  PROC DrawPart23()
    MoveL Offs(pOrigin,99.71,-142.38,-0.00),v40,z0,tcp\WObj:=Plywood;
    MoveL Offs(pOrigin,98.01,-141.25,-0.00),v40,z0,tcp\WObj:=Plywood;
    MoveL Offs(pOrigin,101.27,-145.36,-0.00),v40,fine,tcp\WObj:=Plywood;
    MoveL Offs(pOrigin,101.27,-145.36,-6.00),v60,z5,tcp\WObj:=Plywood;
    MoveL Offs(pOrigin,101.48,-143.34,-6.00),vTravel,z5,tcp\WObj:=Plywood;
    MoveL Offs(pOrigin,101.48,-143.34,-0.00),v60,z0,tcp\WObj:=Plywood;
    MoveL Offs(pOrigin,101.02,-141.85,-0.00),v40,z0,tcp\WObj:=Plywood;
    MoveL Offs(pOrigin,99.39,-139.44,-0.00),v40,z0,tcp\WObj:=Plywood;
    MoveL Offs(pOrigin,99.36,-140.36,-0.00),v40,z0,tcp\WObj:=Plywood;
    MoveL Offs(pOrigin,101.48,-143.34,-0.00),v40,fine,tcp\WObj:=Plywood;
    MoveL Offs(pOrigin,101.48,-143.34,-6.00),v60,z5,tcp\WObj:=Plywood;
    MoveL Offs(pOrigin,99.15,-144.93,-6.00),vTravel,z5,tcp\WObj:=Plywood;
    MoveL Offs(pOrigin,99.15,-144.93,-0.00),v60,z0,tcp\WObj:=Plywood;
    MoveL Offs(pOrigin,97.91,-143.34,-0.00),v40,z0,tcp\WObj:=Plywood;
    MoveL Offs(pOrigin,97.06,-142.95,-0.00),v40,z0,tcp\WObj:=Plywood;
    MoveL Offs(pOrigin,99.15,-144.93,-0.00),v40,fine,tcp\WObj:=Plywood;
    MoveL Offs(pOrigin,99.15,-144.93,-6.00),v60,z5,tcp\WObj:=Plywood;
    MoveL Offs(pOrigin,98.33,-142.70,-6.00),vTravel,z5,tcp\WObj:=Plywood;
    MoveL Offs(pOrigin,98.33,-142.70,-0.00),v60,z0,tcp\WObj:=Plywood;
    MoveL Offs(pOrigin,98.12,-142.17,-0.00),v40,z0,tcp\WObj:=Plywood;
    MoveL Offs(pOrigin,98.33,-142.70,-0.00),v40,fine,tcp\WObj:=Plywood;
    MoveL Offs(pOrigin,98.33,-142.70,-6.00),v60,z5,tcp\WObj:=Plywood;
    MoveL Offs(pOrigin,97.73,-140.68,-6.00),vTravel,z5,tcp\WObj:=Plywood;
    MoveL Offs(pOrigin,97.73,-140.68,-0.00),v60,z0,tcp\WObj:=Plywood;
    MoveL Offs(pOrigin,98.37,-140.79,-0.00),v40,z0,tcp\WObj:=Plywood;
    MoveL Offs(pOrigin,97.73,-140.68,-0.00),v40,fine,tcp\WObj:=Plywood;
    MoveL Offs(pOrigin,97.73,-140.68,-6.00),v60,z5,tcp\WObj:=Plywood;
    MoveL Offs(pOrigin,98.97,-140.33,-6.00),vTravel,z5,tcp\WObj:=Plywood;
    MoveL Offs(pOrigin,98.97,-140.33,-0.00),v60,z0,tcp\WObj:=Plywood;
    MoveL Offs(pOrigin,98.65,-139.87,-0.00),v40,z0,tcp\WObj:=Plywood;
    MoveL Offs(pOrigin,98.97,-140.33,-0.00),v40,fine,tcp\WObj:=Plywood;
    MoveL Offs(pOrigin,98.97,-140.33,-6.00),v60,z5,tcp\WObj:=Plywood;
    MoveL Offs(pOrigin,99.89,-138.98,-6.00),vTravel,z5,tcp\WObj:=Plywood;
    MoveL Offs(pOrigin,99.89,-138.98,-0.00),v60,z0,tcp\WObj:=Plywood;
    MoveL Offs(pOrigin,100.53,-139.62,-0.00),v40,z0,tcp\WObj:=Plywood;
    MoveL Offs(pOrigin,99.43,-137.71,-0.00),v40,z0,tcp\WObj:=Plywood;
    MoveL Offs(pOrigin,99.89,-138.98,-0.00),v40,z0,tcp\WObj:=Plywood;
    MoveL Offs(pOrigin,100.35,-137.95,-0.00),v40,z0,tcp\WObj:=Plywood;
    MoveL Offs(pOrigin,100.14,-137.35,-0.00),v40,z0,tcp\WObj:=Plywood;
    MoveL Offs(pOrigin,100.35,-137.95,-0.00),v40,fine,tcp\WObj:=Plywood;
    MoveL Offs(pOrigin,100.35,-137.95,-6.00),v60,z5,tcp\WObj:=Plywood;
    MoveL Offs(pOrigin,101.41,-137.18,-6.00),vTravel,z5,tcp\WObj:=Plywood;
    MoveL Offs(pOrigin,101.41,-137.18,-0.00),v60,z0,tcp\WObj:=Plywood;
    MoveL Offs(pOrigin,101.84,-137.95,-0.00),v40,z0,tcp\WObj:=Plywood;
    MoveL Offs(pOrigin,101.41,-136.18,-0.00),v40,z0,tcp\WObj:=Plywood;
    MoveL Offs(pOrigin,101.41,-137.18,-0.00),v40,z0,tcp\WObj:=Plywood;
    MoveL Offs(pOrigin,100.88,-136.57,-0.00),v40,z0,tcp\WObj:=Plywood;
    MoveL Offs(pOrigin,100.92,-136.22,-0.00),v40,z0,tcp\WObj:=Plywood;
    MoveL Offs(pOrigin,100.56,-136.04,-0.00),v40,z0,tcp\WObj:=Plywood;
    MoveL Offs(pOrigin,100.88,-136.57,-0.00),v40,z0,tcp\WObj:=Plywood;
    MoveL Offs(pOrigin,100.99,-136.01,-0.00),v40,z0,tcp\WObj:=Plywood;
    MoveL Offs(pOrigin,100.78,-135.58,-0.00),v40,z0,tcp\WObj:=Plywood;
    MoveL Offs(pOrigin,100.99,-136.01,-0.00),v40,z0,tcp\WObj:=Plywood;
    MoveL Offs(pOrigin,100.56,-135.05,-0.00),v40,z0,tcp\WObj:=Plywood;
    MoveL Offs(pOrigin,100.99,-135.26,-0.00),v40,z0,tcp\WObj:=Plywood;
    MoveL Offs(pOrigin,100.56,-135.05,-0.00),v40,fine,tcp\WObj:=Plywood;
    MoveL Offs(pOrigin,100.56,-135.05,-6.00),v60,z5,tcp\WObj:=Plywood;
    MoveL Offs(pOrigin,102.05,-133.99,-6.00),vTravel,z5,tcp\WObj:=Plywood;
    MoveL Offs(pOrigin,102.05,-133.99,-0.00),v60,z0,tcp\WObj:=Plywood;
    MoveL Offs(pOrigin,103.32,-134.34,-0.00),v40,z0,tcp\WObj:=Plywood;
    MoveL Offs(pOrigin,103.93,-134.94,-0.00),v40,z0,tcp\WObj:=Plywood;
    MoveL Offs(pOrigin,103.54,-132.54,-0.00),v40,z0,tcp\WObj:=Plywood;
    MoveL Offs(pOrigin,102.90,-133.17,-0.00),v40,z0,tcp\WObj:=Plywood;
    MoveL Offs(pOrigin,101.84,-133.03,-0.00),v40,z0,tcp\WObj:=Plywood;
    MoveL Offs(pOrigin,101.73,-133.56,-0.00),v40,z0,tcp\WObj:=Plywood;
    MoveL Offs(pOrigin,102.05,-133.99,-0.00),v40,fine,tcp\WObj:=Plywood;
    MoveL Offs(pOrigin,102.05,-133.99,-6.00),v60,z5,tcp\WObj:=Plywood;
    MoveL Offs(pOrigin,103.86,-134.20,-6.00),vTravel,z5,tcp\WObj:=Plywood;
    MoveL Offs(pOrigin,103.86,-134.20,-0.00),v60,z0,tcp\WObj:=Plywood;
    MoveL Offs(pOrigin,104.60,-135.37,-0.00),v40,z0,tcp\WObj:=Plywood;
    MoveL Offs(pOrigin,109.38,-136.86,-0.00),v40,z0,tcp\WObj:=Plywood;
    MoveL Offs(pOrigin,112.14,-137.18,-0.00),v40,z0,tcp\WObj:=Plywood;
    MoveL Offs(pOrigin,116.07,-137.07,-0.00),v40,z0,tcp\WObj:=Plywood;
    MoveL Offs(pOrigin,117.35,-136.68,-0.00),v40,z0,tcp\WObj:=Plywood;
    MoveL Offs(pOrigin,118.41,-135.62,-0.00),v40,z0,tcp\WObj:=Plywood;
    MoveL Offs(pOrigin,120.86,-136.32,-0.00),v40,z0,tcp\WObj:=Plywood;
    MoveL Offs(pOrigin,122.66,-136.25,-0.00),v40,z0,tcp\WObj:=Plywood;
    MoveL Offs(pOrigin,123.51,-137.71,-0.00),v40,z0,tcp\WObj:=Plywood;
    MoveL Offs(pOrigin,126.06,-138.88,-0.00),v40,z0,tcp\WObj:=Plywood;
    MoveL Offs(pOrigin,132.01,-139.94,-0.00),v40,z0,tcp\WObj:=Plywood;
    MoveL Offs(pOrigin,136.48,-139.44,-0.00),v40,z0,tcp\WObj:=Plywood;
    MoveL Offs(pOrigin,137.22,-138.98,-0.00),v40,z0,tcp\WObj:=Plywood;
    MoveL Offs(pOrigin,137.86,-137.60,-0.00),v40,z0,tcp\WObj:=Plywood;
    MoveL Offs(pOrigin,138.07,-133.77,-0.00),v40,z0,tcp\WObj:=Plywood;
    MoveL Offs(pOrigin,137.32,-131.65,-0.00),v40,z0,tcp\WObj:=Plywood;
    MoveL Offs(pOrigin,134.88,-130.48,-0.00),v40,z0,tcp\WObj:=Plywood;
    MoveL Offs(pOrigin,131.91,-129.84,-0.00),v40,z0,tcp\WObj:=Plywood;
    MoveL Offs(pOrigin,127.55,-129.63,-0.00),v40,z0,tcp\WObj:=Plywood;
    MoveL Offs(pOrigin,126.06,-130.02,-0.00),v40,z0,tcp\WObj:=Plywood;
    MoveL Offs(pOrigin,124.89,-131.01,-0.00),v40,z0,tcp\WObj:=Plywood;
    MoveL Offs(pOrigin,123.90,-132.50,-0.00),v40,z0,tcp\WObj:=Plywood;
    MoveL Offs(pOrigin,122.77,-135.48,-0.00),v40,z0,tcp\WObj:=Plywood;
    MoveL Offs(pOrigin,121.71,-135.79,-0.00),v40,z0,tcp\WObj:=Plywood;
    MoveL Offs(pOrigin,119.79,-135.58,-0.00),v40,z0,tcp\WObj:=Plywood;
    MoveL Offs(pOrigin,118.55,-134.94,-0.00),v40,z0,tcp\WObj:=Plywood;
    MoveL Offs(pOrigin,118.20,-131.44,-0.00),v40,z0,tcp\WObj:=Plywood;
    MoveL Offs(pOrigin,117.49,-129.63,-0.00),v40,z0,tcp\WObj:=Plywood;
    MoveL Offs(pOrigin,116.71,-128.78,-0.00),v40,z0,tcp\WObj:=Plywood;
    MoveL Offs(pOrigin,112.89,-127.61,-0.00),v40,z0,tcp\WObj:=Plywood;
    MoveL Offs(pOrigin,108.53,-127.29,-0.00),v40,z0,tcp\WObj:=Plywood;
    MoveL Offs(pOrigin,106.19,-127.68,-0.00),v40,z0,tcp\WObj:=Plywood;
    MoveL Offs(pOrigin,105.34,-128.36,-0.00),v40,z0,tcp\WObj:=Plywood;
    MoveL Offs(pOrigin,104.56,-129.74,-0.00),v40,z0,tcp\WObj:=Plywood;
    MoveL Offs(pOrigin,103.86,-132.39,-0.00),v40,z0,tcp\WObj:=Plywood;
    MoveL Offs(pOrigin,103.86,-134.20,-0.00),v40,fine,tcp\WObj:=Plywood;
    MoveL Offs(pOrigin,103.86,-134.20,-6.00),v60,z5,tcp\WObj:=Plywood;
    MoveL Offs(pOrigin,106.44,-133.85,-6.00),vTravel,z5,tcp\WObj:=Plywood;
    MoveL Offs(pOrigin,106.44,-133.85,-0.00),v60,z0,tcp\WObj:=Plywood;
    MoveL Offs(pOrigin,107.79,-135.19,-0.00),v40,z0,tcp\WObj:=Plywood;
    MoveL Offs(pOrigin,110.44,-136.11,-0.00),v40,z0,tcp\WObj:=Plywood;
    MoveL Offs(pOrigin,115.22,-136.54,-0.00),v40,z0,tcp\WObj:=Plywood;
    MoveL Offs(pOrigin,117.24,-136.01,-0.00),v40,z0,tcp\WObj:=Plywood;
    MoveL Offs(pOrigin,117.67,-134.98,-0.00),v40,z0,tcp\WObj:=Plywood;
    MoveL Offs(pOrigin,117.24,-135.16,-0.00),v40,z0,tcp\WObj:=Plywood;
    MoveL Offs(pOrigin,117.35,-134.77,-0.00),v40,z0,tcp\WObj:=Plywood;
    MoveL Offs(pOrigin,115.22,-135.69,-0.00),v40,z0,tcp\WObj:=Plywood;
    MoveL Offs(pOrigin,112.46,-135.48,-0.00),v40,z0,tcp\WObj:=Plywood;
    MoveL Offs(pOrigin,109.81,-134.45,-0.00),v40,z0,tcp\WObj:=Plywood;
    MoveL Offs(pOrigin,107.75,-132.39,-0.00),v40,z0,tcp\WObj:=Plywood;
    MoveL Offs(pOrigin,108.43,-132.64,-0.00),v40,z0,tcp\WObj:=Plywood;
  ENDPROC

  PROC DrawPart24()
    MoveL Offs(pOrigin,108.32,-132.29,-0.00),v40,z0,tcp\WObj:=Plywood;
    MoveL Offs(pOrigin,106.48,-131.76,-0.00),v40,z0,tcp\WObj:=Plywood;
    MoveL Offs(pOrigin,108.00,-131.86,-0.00),v40,z0,tcp\WObj:=Plywood;
    MoveL Offs(pOrigin,110.12,-132.82,-0.00),v40,z0,tcp\WObj:=Plywood;
    MoveL Offs(pOrigin,112.68,-132.61,-0.00),v40,z0,tcp\WObj:=Plywood;
    MoveL Offs(pOrigin,117.46,-133.46,-0.00),v40,z0,tcp\WObj:=Plywood;
    MoveL Offs(pOrigin,115.01,-134.77,-0.00),v40,z0,tcp\WObj:=Plywood;
    MoveL Offs(pOrigin,113.21,-135.05,-0.00),v40,z0,tcp\WObj:=Plywood;
    MoveL Offs(pOrigin,110.76,-134.34,-0.00),v40,z0,tcp\WObj:=Plywood;
    MoveL Offs(pOrigin,108.99,-133.03,-0.00),v40,z0,tcp\WObj:=Plywood;
    MoveL Offs(pOrigin,110.23,-134.45,-0.00),v40,z0,tcp\WObj:=Plywood;
    MoveL Offs(pOrigin,113.10,-135.48,-0.00),v40,z0,tcp\WObj:=Plywood;
    MoveL Offs(pOrigin,115.01,-135.30,-0.00),v40,z0,tcp\WObj:=Plywood;
    MoveL Offs(pOrigin,117.35,-134.34,-0.00),v40,z0,tcp\WObj:=Plywood;
    MoveL Offs(pOrigin,117.88,-133.77,-0.00),v40,z0,tcp\WObj:=Plywood;
    MoveL Offs(pOrigin,116.39,-131.65,-0.00),v40,z0,tcp\WObj:=Plywood;
    MoveL Offs(pOrigin,114.55,-130.13,-0.00),v40,z0,tcp\WObj:=Plywood;
    MoveL Offs(pOrigin,115.76,-130.80,-0.00),v40,z0,tcp\WObj:=Plywood;
    MoveL Offs(pOrigin,117.24,-132.43,-0.00),v40,z0,tcp\WObj:=Plywood;
    MoveL Offs(pOrigin,117.70,-131.40,-0.00),v40,z0,tcp\WObj:=Plywood;
    MoveL Offs(pOrigin,117.99,-132.29,-0.00),v40,z0,tcp\WObj:=Plywood;
    MoveL Offs(pOrigin,118.09,-134.41,-0.00),v40,z0,tcp\WObj:=Plywood;
    MoveL Offs(pOrigin,117.81,-135.48,-0.00),v40,z0,tcp\WObj:=Plywood;
    MoveL Offs(pOrigin,117.35,-136.11,-0.00),v40,z0,tcp\WObj:=Plywood;
    MoveL Offs(pOrigin,116.29,-136.54,-0.00),v40,z0,tcp\WObj:=Plywood;
    MoveL Offs(pOrigin,111.93,-136.64,-0.00),v40,z0,tcp\WObj:=Plywood;
    MoveL Offs(pOrigin,108.74,-136.22,-0.00),v40,z0,tcp\WObj:=Plywood;
    MoveL Offs(pOrigin,106.94,-135.58,-0.00),v40,z0,tcp\WObj:=Plywood;
    MoveL Offs(pOrigin,106.48,-134.62,-0.00),v40,z0,tcp\WObj:=Plywood;
    MoveL Offs(pOrigin,106.44,-133.85,-0.00),v40,fine,tcp\WObj:=Plywood;
    MoveL Offs(pOrigin,106.44,-133.85,-6.00),v60,z5,tcp\WObj:=Plywood;
    MoveL Offs(pOrigin,110.37,-133.35,-6.00),vTravel,z5,tcp\WObj:=Plywood;
    MoveL Offs(pOrigin,110.37,-133.35,-0.00),v60,z0,tcp\WObj:=Plywood;
    MoveL Offs(pOrigin,111.40,-134.06,-0.00),v40,z0,tcp\WObj:=Plywood;
    MoveL Offs(pOrigin,112.14,-132.82,-0.00),v40,z0,tcp\WObj:=Plywood;
    MoveL Offs(pOrigin,110.87,-132.82,-0.00),v40,z0,tcp\WObj:=Plywood;
    MoveL Offs(pOrigin,110.37,-133.35,-0.00),v40,fine,tcp\WObj:=Plywood;
    MoveL Offs(pOrigin,110.37,-133.35,-6.00),v60,z5,tcp\WObj:=Plywood;
    MoveL Offs(pOrigin,112.29,-134.31,-6.00),vTravel,z5,tcp\WObj:=Plywood;
    MoveL Offs(pOrigin,112.29,-134.31,-0.00),v60,z0,tcp\WObj:=Plywood;
    MoveL Offs(pOrigin,112.68,-134.48,-0.00),v40,z0,tcp\WObj:=Plywood;
    MoveL Offs(pOrigin,112.85,-134.20,-0.00),v40,z0,tcp\WObj:=Plywood;
    MoveL Offs(pOrigin,112.57,-133.99,-0.00),v40,z0,tcp\WObj:=Plywood;
    MoveL Offs(pOrigin,112.29,-134.31,-0.00),v40,fine,tcp\WObj:=Plywood;
    MoveL Offs(pOrigin,112.29,-134.31,-6.00),v60,z5,tcp\WObj:=Plywood;
    MoveL Offs(pOrigin,114.38,-133.24,-6.00),vTravel,z5,tcp\WObj:=Plywood;
    MoveL Offs(pOrigin,114.38,-133.24,-0.00),v60,z0,tcp\WObj:=Plywood;
    MoveL Offs(pOrigin,114.69,-134.38,-0.00),v40,z0,tcp\WObj:=Plywood;
    MoveL Offs(pOrigin,115.93,-133.77,-0.00),v40,z0,tcp\WObj:=Plywood;
    MoveL Offs(pOrigin,114.38,-133.24,-0.00),v40,fine,tcp\WObj:=Plywood;
    MoveL Offs(pOrigin,114.38,-133.24,-6.00),v60,z5,tcp\WObj:=Plywood;
    MoveL Offs(pOrigin,116.43,-132.25,-6.00),vTravel,z5,tcp\WObj:=Plywood;
    MoveL Offs(pOrigin,116.43,-132.25,-0.00),v60,z0,tcp\WObj:=Plywood;
    MoveL Offs(pOrigin,112.00,-130.80,-0.00),v40,z0,tcp\WObj:=Plywood;
    MoveL Offs(pOrigin,116.43,-132.25,-0.00),v40,z0,tcp\WObj:=Plywood;
    MoveL Offs(pOrigin,117.46,-132.50,-0.00),v40,z0,tcp\WObj:=Plywood;
    MoveL Offs(pOrigin,117.78,-132.89,-0.00),v40,z0,tcp\WObj:=Plywood;
    MoveL Offs(pOrigin,117.67,-132.29,-0.00),v40,z0,tcp\WObj:=Plywood;
    MoveL Offs(pOrigin,117.46,-132.50,-0.00),v40,fine,tcp\WObj:=Plywood;
    MoveL Offs(pOrigin,117.46,-132.50,-6.00),v60,z5,tcp\WObj:=Plywood;
    MoveL Offs(pOrigin,118.84,-133.35,-6.00),vTravel,z5,tcp\WObj:=Plywood;
    MoveL Offs(pOrigin,118.84,-133.35,-0.00),v60,z0,tcp\WObj:=Plywood;
    MoveL Offs(pOrigin,118.73,-132.82,-0.00),v40,z0,tcp\WObj:=Plywood;
    MoveL Offs(pOrigin,118.84,-133.35,-0.00),v40,fine,tcp\WObj:=Plywood;
    MoveL Offs(pOrigin,118.84,-133.35,-6.00),v60,z5,tcp\WObj:=Plywood;
    MoveL Offs(pOrigin,118.09,-136.96,-6.00),vTravel,z5,tcp\WObj:=Plywood;
    MoveL Offs(pOrigin,118.09,-136.96,-0.00),v60,z0,tcp\WObj:=Plywood;
    MoveL Offs(pOrigin,118.20,-136.43,-0.00),v40,z0,tcp\WObj:=Plywood;
    MoveL Offs(pOrigin,118.09,-136.96,-0.00),v40,fine,tcp\WObj:=Plywood;
    MoveL Offs(pOrigin,118.09,-136.96,-6.00),v60,z5,tcp\WObj:=Plywood;
    MoveL Offs(pOrigin,123.37,-136.75,-6.00),vTravel,z5,tcp\WObj:=Plywood;
    MoveL Offs(pOrigin,123.37,-136.75,-0.00),v60,z0,tcp\WObj:=Plywood;
    MoveL Offs(pOrigin,123.30,-135.16,-0.00),v40,z0,tcp\WObj:=Plywood;
    MoveL Offs(pOrigin,124.29,-132.71,-0.00),v40,z0,tcp\WObj:=Plywood;
    MoveL Offs(pOrigin,125.00,-132.36,-0.00),v40,z0,tcp\WObj:=Plywood;
    MoveL Offs(pOrigin,124.82,-133.46,-0.00),v40,z0,tcp\WObj:=Plywood;
    MoveL Offs(pOrigin,123.41,-135.37,-0.00),v40,z0,tcp\WObj:=Plywood;
    MoveL Offs(pOrigin,123.48,-136.64,-0.00),v40,z0,tcp\WObj:=Plywood;
    MoveL Offs(pOrigin,124.47,-137.67,-0.00),v40,z0,tcp\WObj:=Plywood;
    MoveL Offs(pOrigin,132.01,-138.98,-0.00),v40,z0,tcp\WObj:=Plywood;
    MoveL Offs(pOrigin,135.41,-138.45,-0.00),v40,z0,tcp\WObj:=Plywood;
    MoveL Offs(pOrigin,134.46,-139.30,-0.00),v40,z0,tcp\WObj:=Plywood;
    MoveL Offs(pOrigin,131.80,-139.41,-0.00),v40,z0,tcp\WObj:=Plywood;
    MoveL Offs(pOrigin,125.21,-138.06,-0.00),v40,z0,tcp\WObj:=Plywood;
    MoveL Offs(pOrigin,123.37,-136.75,-0.00),v40,fine,tcp\WObj:=Plywood;
    MoveL Offs(pOrigin,123.37,-136.75,-6.00),v60,z5,tcp\WObj:=Plywood;
    MoveL Offs(pOrigin,124.40,-135.86,-6.00),vTravel,z5,tcp\WObj:=Plywood;
    MoveL Offs(pOrigin,124.40,-135.86,-0.00),v60,z0,tcp\WObj:=Plywood;
    MoveL Offs(pOrigin,124.26,-135.37,-0.00),v40,z0,tcp\WObj:=Plywood;
    MoveL Offs(pOrigin,124.61,-135.16,-0.00),v40,z0,tcp\WObj:=Plywood;
    MoveL Offs(pOrigin,124.54,-134.38,-0.00),v40,z0,tcp\WObj:=Plywood;
    MoveL Offs(pOrigin,124.79,-134.94,-0.00),v40,z0,tcp\WObj:=Plywood;
    MoveL Offs(pOrigin,126.91,-136.75,-0.00),v40,z0,tcp\WObj:=Plywood;
    MoveL Offs(pOrigin,128.72,-137.39,-0.00),v40,z0,tcp\WObj:=Plywood;
    MoveL Offs(pOrigin,131.48,-137.28,-0.00),v40,z0,tcp\WObj:=Plywood;
    MoveL Offs(pOrigin,132.86,-136.89,-0.00),v40,z0,tcp\WObj:=Plywood;
    MoveL Offs(pOrigin,133.46,-136.32,-0.00),v40,z0,tcp\WObj:=Plywood;
    MoveL Offs(pOrigin,130.74,-137.07,-0.00),v40,z0,tcp\WObj:=Plywood;
    MoveL Offs(pOrigin,129.25,-136.96,-0.00),v40,z0,tcp\WObj:=Plywood;
    MoveL Offs(pOrigin,127.12,-136.01,-0.00),v40,z0,tcp\WObj:=Plywood;
    MoveL Offs(pOrigin,125.43,-134.73,-0.00),v40,z0,tcp\WObj:=Plywood;
    MoveL Offs(pOrigin,125.35,-134.34,-0.00),v40,z0,tcp\WObj:=Plywood;
    MoveL Offs(pOrigin,130.95,-134.84,-0.00),v40,z0,tcp\WObj:=Plywood;
    MoveL Offs(pOrigin,131.80,-136.32,-0.00),v40,z0,tcp\WObj:=Plywood;
    MoveL Offs(pOrigin,132.65,-135.79,-0.00),v40,z0,tcp\WObj:=Plywood;
    MoveL Offs(pOrigin,131.69,-135.05,-0.00),v40,z0,tcp\WObj:=Plywood;
    MoveL Offs(pOrigin,132.86,-135.48,-0.00),v40,z0,tcp\WObj:=Plywood;
    MoveL Offs(pOrigin,135.20,-135.19,-0.00),v40,z0,tcp\WObj:=Plywood;
    MoveL Offs(pOrigin,136.30,-135.48,-0.00),v40,z0,tcp\WObj:=Plywood;
    MoveL Offs(pOrigin,134.56,-135.62,-0.00),v40,z0,tcp\WObj:=Plywood;
    MoveL Offs(pOrigin,134.35,-135.97,-0.00),v40,z0,tcp\WObj:=Plywood;
    MoveL Offs(pOrigin,135.24,-135.83,-0.00),v40,z0,tcp\WObj:=Plywood;
    MoveL Offs(pOrigin,132.65,-137.18,-0.00),v40,z0,tcp\WObj:=Plywood;
    MoveL Offs(pOrigin,128.82,-137.60,-0.00),v40,z0,tcp\WObj:=Plywood;
    MoveL Offs(pOrigin,126.91,-137.25,-0.00),v40,z0,tcp\WObj:=Plywood;
    MoveL Offs(pOrigin,124.68,-135.55,-0.00),v40,z0,tcp\WObj:=Plywood;
    MoveL Offs(pOrigin,124.40,-135.86,-0.00),v40,z0,tcp\WObj:=Plywood;
    MoveL Offs(pOrigin,125.32,-135.65,-0.00),v40,z0,tcp\WObj:=Plywood;
    MoveL Offs(pOrigin,124.68,-135.19,-0.00),v40,z0,tcp\WObj:=Plywood;
    MoveL Offs(pOrigin,125.32,-135.65,-0.00),v40,fine,tcp\WObj:=Plywood;
  ENDPROC

  PROC DrawPart25()
    MoveL Offs(pOrigin,125.32,-135.65,-6.00),v60,z5,tcp\WObj:=Plywood;
    MoveL Offs(pOrigin,126.98,-135.16,-6.00),vTravel,z5,tcp\WObj:=Plywood;
    MoveL Offs(pOrigin,126.98,-135.16,-0.00),v60,z0,tcp\WObj:=Plywood;
    MoveL Offs(pOrigin,128.19,-136.11,-0.00),v40,z0,tcp\WObj:=Plywood;
    MoveL Offs(pOrigin,129.00,-134.84,-0.00),v40,z0,tcp\WObj:=Plywood;
    MoveL Offs(pOrigin,127.23,-134.84,-0.00),v40,z0,tcp\WObj:=Plywood;
    MoveL Offs(pOrigin,126.98,-135.16,-0.00),v40,fine,tcp\WObj:=Plywood;
    MoveL Offs(pOrigin,126.98,-135.16,-6.00),v60,z5,tcp\WObj:=Plywood;
    MoveL Offs(pOrigin,127.09,-133.49,-6.00),vTravel,z5,tcp\WObj:=Plywood;
    MoveL Offs(pOrigin,127.09,-133.49,-0.00),v60,z0,tcp\WObj:=Plywood;
    MoveL Offs(pOrigin,128.75,-133.14,-0.00),v40,z0,tcp\WObj:=Plywood;
    MoveL Offs(pOrigin,127.09,-133.49,-0.00),v40,fine,tcp\WObj:=Plywood;
    MoveL Offs(pOrigin,127.09,-133.49,-6.00),v60,z5,tcp\WObj:=Plywood;
    MoveL Offs(pOrigin,125.89,-133.31,-6.00),vTravel,z5,tcp\WObj:=Plywood;
    MoveL Offs(pOrigin,125.89,-133.31,-0.00),v60,z0,tcp\WObj:=Plywood;
    MoveL Offs(pOrigin,127.66,-132.25,-0.00),v40,z0,tcp\WObj:=Plywood;
    MoveL Offs(pOrigin,129.92,-131.76,-0.00),v40,z0,tcp\WObj:=Plywood;
    MoveL Offs(pOrigin,125.89,-133.31,-0.00),v40,z0,tcp\WObj:=Plywood;
    MoveL Offs(pOrigin,124.72,-133.24,-0.00),v40,z0,tcp\WObj:=Plywood;
    MoveL Offs(pOrigin,124.57,-132.96,-0.00),v40,z0,tcp\WObj:=Plywood;
    MoveL Offs(pOrigin,124.26,-133.63,-0.00),v40,z0,tcp\WObj:=Plywood;
    MoveL Offs(pOrigin,124.72,-133.24,-0.00),v40,fine,tcp\WObj:=Plywood;
    MoveL Offs(pOrigin,124.72,-133.24,-6.00),v60,z5,tcp\WObj:=Plywood;
    MoveL Offs(pOrigin,123.83,-134.27,-6.00),vTravel,z5,tcp\WObj:=Plywood;
    MoveL Offs(pOrigin,123.83,-134.27,-0.00),v60,z0,tcp\WObj:=Plywood;
    MoveL Offs(pOrigin,124.04,-133.81,-0.00),v40,z0,tcp\WObj:=Plywood;
    MoveL Offs(pOrigin,123.83,-134.27,-0.00),v40,fine,tcp\WObj:=Plywood;
    MoveL Offs(pOrigin,123.83,-134.27,-6.00),v60,z5,tcp\WObj:=Plywood;
    MoveL Offs(pOrigin,123.55,-138.73,-6.00),vTravel,z5,tcp\WObj:=Plywood;
    MoveL Offs(pOrigin,123.55,-138.73,-0.00),v60,z0,tcp\WObj:=Plywood;
    MoveL Offs(pOrigin,124.22,-140.08,-0.00),v40,z0,tcp\WObj:=Plywood;
    MoveL Offs(pOrigin,123.69,-139.51,-0.00),v40,z0,tcp\WObj:=Plywood;
    MoveL Offs(pOrigin,123.55,-138.73,-0.00),v40,fine,tcp\WObj:=Plywood;
    MoveL Offs(pOrigin,123.55,-138.73,-6.00),v60,z5,tcp\WObj:=Plywood;
    MoveL Offs(pOrigin,129.14,-136.32,-6.00),vTravel,z5,tcp\WObj:=Plywood;
    MoveL Offs(pOrigin,129.14,-136.32,-0.00),v60,z0,tcp\WObj:=Plywood;
    MoveL Offs(pOrigin,129.75,-136.43,-0.00),v40,z0,tcp\WObj:=Plywood;
    MoveL Offs(pOrigin,129.36,-136.11,-0.00),v40,z0,tcp\WObj:=Plywood;
    MoveL Offs(pOrigin,129.14,-136.32,-0.00),v40,fine,tcp\WObj:=Plywood;
    MoveL Offs(pOrigin,129.14,-136.32,-6.00),v60,z5,tcp\WObj:=Plywood;
    MoveL Offs(pOrigin,127.30,-127.90,-6.00),vTravel,z5,tcp\WObj:=Plywood;
    MoveL Offs(pOrigin,127.30,-127.90,-0.00),v60,z0,tcp\WObj:=Plywood;
    MoveL Offs(pOrigin,128.08,-126.23,-0.00),v40,z0,tcp\WObj:=Plywood;
    MoveL Offs(pOrigin,127.62,-124.85,-0.00),v40,z0,tcp\WObj:=Plywood;
    MoveL Offs(pOrigin,126.91,-124.35,-0.00),v40,z0,tcp\WObj:=Plywood;
    MoveL Offs(pOrigin,126.28,-124.74,-0.00),v40,z0,tcp\WObj:=Plywood;
    MoveL Offs(pOrigin,125.21,-124.57,-0.00),v40,z0,tcp\WObj:=Plywood;
    MoveL Offs(pOrigin,122.98,-122.62,-0.00),v40,z0,tcp\WObj:=Plywood;
    MoveL Offs(pOrigin,122.13,-122.30,-0.00),v40,z0,tcp\WObj:=Plywood;
    MoveL Offs(pOrigin,120.96,-122.37,-0.00),v40,z0,tcp\WObj:=Plywood;
    MoveL Offs(pOrigin,118.73,-123.68,-0.00),v40,z0,tcp\WObj:=Plywood;
    MoveL Offs(pOrigin,117.24,-123.26,-0.00),v40,z0,tcp\WObj:=Plywood;
    MoveL Offs(pOrigin,116.61,-123.57,-0.00),v40,z0,tcp\WObj:=Plywood;
    MoveL Offs(pOrigin,116.07,-125.06,-0.00),v40,z0,tcp\WObj:=Plywood;
    MoveL Offs(pOrigin,116.64,-126.73,-0.00),v40,z0,tcp\WObj:=Plywood;
    MoveL Offs(pOrigin,115.97,-125.38,-0.00),v40,z0,tcp\WObj:=Plywood;
    MoveL Offs(pOrigin,116.29,-123.68,-0.00),v40,z0,tcp\WObj:=Plywood;
    MoveL Offs(pOrigin,117.24,-123.04,-0.00),v40,z0,tcp\WObj:=Plywood;
    MoveL Offs(pOrigin,119.05,-123.15,-0.00),v40,z0,tcp\WObj:=Plywood;
    MoveL Offs(pOrigin,119.86,-122.62,-0.00),v40,z0,tcp\WObj:=Plywood;
    MoveL Offs(pOrigin,118.62,-122.62,-0.00),v40,z0,tcp\WObj:=Plywood;
    MoveL Offs(pOrigin,117.35,-121.84,-0.00),v40,z0,tcp\WObj:=Plywood;
    MoveL Offs(pOrigin,117.24,-122.16,-0.00),v40,z0,tcp\WObj:=Plywood;
    MoveL Offs(pOrigin,116.18,-121.38,-0.00),v40,z0,tcp\WObj:=Plywood;
    MoveL Offs(pOrigin,115.86,-121.63,-0.00),v40,z0,tcp\WObj:=Plywood;
    MoveL Offs(pOrigin,115.22,-120.32,-0.00),v40,z0,tcp\WObj:=Plywood;
    MoveL Offs(pOrigin,115.01,-121.06,-0.00),v40,z0,tcp\WObj:=Plywood;
    MoveL Offs(pOrigin,112.36,-119.93,-0.00),v40,z0,tcp\WObj:=Plywood;
    MoveL Offs(pOrigin,111.86,-119.32,-0.00),v40,z0,tcp\WObj:=Plywood;
    MoveL Offs(pOrigin,111.61,-117.73,-0.00),v40,z0,tcp\WObj:=Plywood;
    MoveL Offs(pOrigin,111.90,-116.78,-0.00),v40,z0,tcp\WObj:=Plywood;
    MoveL Offs(pOrigin,112.46,-116.24,-0.00),v40,z0,tcp\WObj:=Plywood;
    MoveL Offs(pOrigin,113.74,-115.82,-0.00),v40,z0,tcp\WObj:=Plywood;
    MoveL Offs(pOrigin,114.27,-116.63,-0.00),v40,z0,tcp\WObj:=Plywood;
    MoveL Offs(pOrigin,115.33,-117.34,-0.00),v40,z0,tcp\WObj:=Plywood;
    MoveL Offs(pOrigin,116.93,-117.20,-0.00),v40,z0,tcp\WObj:=Plywood;
    MoveL Offs(pOrigin,116.93,-117.59,-0.00),v40,z0,tcp\WObj:=Plywood;
    MoveL Offs(pOrigin,119.79,-118.16,-0.00),v40,z0,tcp\WObj:=Plywood;
    MoveL Offs(pOrigin,123.09,-118.26,-0.00),v40,z0,tcp\WObj:=Plywood;
    MoveL Offs(pOrigin,127.55,-119.11,-0.00),v40,z0,tcp\WObj:=Plywood;
    MoveL Offs(pOrigin,130.52,-119.01,-0.00),v40,z0,tcp\WObj:=Plywood;
    MoveL Offs(pOrigin,131.38,-119.36,-0.00),v40,z0,tcp\WObj:=Plywood;
    MoveL Offs(pOrigin,133.29,-118.86,-0.00),v40,z0,tcp\WObj:=Plywood;
    MoveL Offs(pOrigin,133.71,-118.40,-0.00),v40,z0,tcp\WObj:=Plywood;
    MoveL Offs(pOrigin,134.63,-118.90,-0.00),v40,z0,tcp\WObj:=Plywood;
    MoveL Offs(pOrigin,135.09,-120.28,-0.00),v40,z0,tcp\WObj:=Plywood;
    MoveL Offs(pOrigin,134.53,-121.98,-0.00),v40,z0,tcp\WObj:=Plywood;
    MoveL Offs(pOrigin,132.47,-122.97,-0.00),v40,z0,tcp\WObj:=Plywood;
    MoveL Offs(pOrigin,132.44,-122.58,-0.00),v40,z0,tcp\WObj:=Plywood;
    MoveL Offs(pOrigin,131.59,-123.01,-0.00),v40,z0,tcp\WObj:=Plywood;
    MoveL Offs(pOrigin,130.67,-123.08,-0.00),v40,z0,tcp\WObj:=Plywood;
    MoveL Offs(pOrigin,130.52,-122.76,-0.00),v40,z0,tcp\WObj:=Plywood;
    MoveL Offs(pOrigin,129.92,-123.11,-0.00),v40,z0,tcp\WObj:=Plywood;
    MoveL Offs(pOrigin,129.78,-122.80,-0.00),v40,z0,tcp\WObj:=Plywood;
    MoveL Offs(pOrigin,128.40,-123.40,-0.00),v40,z0,tcp\WObj:=Plywood;
    MoveL Offs(pOrigin,128.51,-122.80,-0.00),v40,z0,tcp\WObj:=Plywood;
    MoveL Offs(pOrigin,127.87,-123.22,-0.00),v40,z0,tcp\WObj:=Plywood;
    MoveL Offs(pOrigin,125.53,-123.57,-0.00),v40,z0,tcp\WObj:=Plywood;
    MoveL Offs(pOrigin,124.79,-123.43,-0.00),v40,z0,tcp\WObj:=Plywood;
    MoveL Offs(pOrigin,123.72,-122.65,-0.00),v40,z0,tcp\WObj:=Plywood;
    MoveL Offs(pOrigin,125.11,-124.04,-0.00),v40,z0,tcp\WObj:=Plywood;
    MoveL Offs(pOrigin,126.17,-124.39,-0.00),v40,z0,tcp\WObj:=Plywood;
    MoveL Offs(pOrigin,126.38,-124.00,-0.00),v40,z0,tcp\WObj:=Plywood;
    MoveL Offs(pOrigin,127.76,-124.64,-0.00),v40,z0,tcp\WObj:=Plywood;
    MoveL Offs(pOrigin,128.29,-126.23,-0.00),v40,z0,tcp\WObj:=Plywood;
    MoveL Offs(pOrigin,128.05,-127.08,-0.00),v40,z0,tcp\WObj:=Plywood;
    MoveL Offs(pOrigin,127.30,-127.90,-0.00),v40,fine,tcp\WObj:=Plywood;
    MoveL Offs(pOrigin,127.30,-127.90,-6.00),v60,z5,tcp\WObj:=Plywood;
    MoveL Offs(pOrigin,128.68,-127.33,-6.00),vTravel,z5,tcp\WObj:=Plywood;
    MoveL Offs(pOrigin,128.68,-127.33,-0.00),v60,z0,tcp\WObj:=Plywood;
    MoveL Offs(pOrigin,134.60,-122.34,-0.00),v40,z0,tcp\WObj:=Plywood;
    MoveL Offs(pOrigin,128.68,-127.33,-0.00),v40,fine,tcp\WObj:=Plywood;
    MoveL Offs(pOrigin,128.68,-127.33,-6.00),v60,z5,tcp\WObj:=Plywood;
    MoveL Offs(pOrigin,127.97,-120.56,-6.00),vTravel,z5,tcp\WObj:=Plywood;
    MoveL Offs(pOrigin,127.97,-120.56,-0.00),v60,z0,tcp\WObj:=Plywood;
    MoveL Offs(pOrigin,130.91,-120.07,-0.00),v40,z0,tcp\WObj:=Plywood;
    MoveL Offs(pOrigin,129.68,-119.43,-0.00),v40,z0,tcp\WObj:=Plywood;
    MoveL Offs(pOrigin,126.38,-119.22,-0.00),v40,z0,tcp\WObj:=Plywood;
    MoveL Offs(pOrigin,123.62,-118.58,-0.00),v40,z0,tcp\WObj:=Plywood;
    MoveL Offs(pOrigin,119.69,-118.37,-0.00),v40,z0,tcp\WObj:=Plywood;
  ENDPROC

  PROC DrawPart26()
    MoveL Offs(pOrigin,117.78,-117.94,-0.00),v40,z0,tcp\WObj:=Plywood;
    MoveL Offs(pOrigin,116.82,-117.98,-0.00),v40,z0,tcp\WObj:=Plywood;
    MoveL Offs(pOrigin,116.96,-118.26,-0.00),v40,z0,tcp\WObj:=Plywood;
    MoveL Offs(pOrigin,115.61,-118.05,-0.00),v40,z0,tcp\WObj:=Plywood;
    MoveL Offs(pOrigin,116.39,-118.76,-0.00),v40,z0,tcp\WObj:=Plywood;
    MoveL Offs(pOrigin,117.88,-119.25,-0.00),v40,z0,tcp\WObj:=Plywood;
    MoveL Offs(pOrigin,118.16,-119.01,-0.00),v40,z0,tcp\WObj:=Plywood;
    MoveL Offs(pOrigin,117.63,-118.65,-0.00),v40,z0,tcp\WObj:=Plywood;
    MoveL Offs(pOrigin,118.70,-119.04,-0.00),v40,z0,tcp\WObj:=Plywood;
    MoveL Offs(pOrigin,118.73,-119.50,-0.00),v40,z0,tcp\WObj:=Plywood;
    MoveL Offs(pOrigin,119.16,-119.22,-0.00),v40,z0,tcp\WObj:=Plywood;
    MoveL Offs(pOrigin,119.16,-119.57,-0.00),v40,z0,tcp\WObj:=Plywood;
    MoveL Offs(pOrigin,121.21,-119.54,-0.00),v40,z0,tcp\WObj:=Plywood;
    MoveL Offs(pOrigin,121.18,-119.96,-0.00),v40,z0,tcp\WObj:=Plywood;
    MoveL Offs(pOrigin,122.41,-120.21,-0.00),v40,z0,tcp\WObj:=Plywood;
    MoveL Offs(pOrigin,122.27,-121.24,-0.00),v40,z0,tcp\WObj:=Plywood;
    MoveL Offs(pOrigin,121.53,-121.88,-0.00),v40,z0,tcp\WObj:=Plywood;
    MoveL Offs(pOrigin,123.19,-122.37,-0.00),v40,z0,tcp\WObj:=Plywood;
    MoveL Offs(pOrigin,123.37,-122.19,-0.00),v40,z0,tcp\WObj:=Plywood;
    MoveL Offs(pOrigin,122.56,-121.13,-0.00),v40,z0,tcp\WObj:=Plywood;
    MoveL Offs(pOrigin,123.09,-120.14,-0.00),v40,z0,tcp\WObj:=Plywood;
    MoveL Offs(pOrigin,123.51,-120.32,-0.00),v40,z0,tcp\WObj:=Plywood;
    MoveL Offs(pOrigin,124.15,-119.86,-0.00),v40,z0,tcp\WObj:=Plywood;
    MoveL Offs(pOrigin,127.62,-120.10,-0.00),v40,z0,tcp\WObj:=Plywood;
    MoveL Offs(pOrigin,127.97,-120.56,-0.00),v40,fine,tcp\WObj:=Plywood;
    MoveL Offs(pOrigin,127.97,-120.56,-6.00),v60,z5,tcp\WObj:=Plywood;
    MoveL Offs(pOrigin,122.41,-114.97,-6.00),vTravel,z5,tcp\WObj:=Plywood;
    MoveL Offs(pOrigin,122.41,-114.97,-0.00),v60,z0,tcp\WObj:=Plywood;
    MoveL Offs(pOrigin,123.12,-115.07,-0.00),v40,z0,tcp\WObj:=Plywood;
    MoveL Offs(pOrigin,122.41,-114.97,-0.00),v40,fine,tcp\WObj:=Plywood;
    MoveL Offs(pOrigin,122.41,-114.97,-6.00),v60,z5,tcp\WObj:=Plywood;
    MoveL Offs(pOrigin,123.94,-106.68,-6.00),vTravel,z5,tcp\WObj:=Plywood;
    MoveL Offs(pOrigin,123.94,-106.68,-0.00),v60,z0,tcp\WObj:=Plywood;
    MoveL Offs(pOrigin,118.94,-106.89,-0.00),v40,z0,tcp\WObj:=Plywood;
    MoveL Offs(pOrigin,114.66,-108.95,-0.00),v40,z0,tcp\WObj:=Plywood;
    MoveL Offs(pOrigin,116.50,-107.60,-0.00),v40,z0,tcp\WObj:=Plywood;
    MoveL Offs(pOrigin,118.94,-106.57,-0.00),v40,z0,tcp\WObj:=Plywood;
    MoveL Offs(pOrigin,123.72,-106.26,-0.00),v40,z0,tcp\WObj:=Plywood;
    MoveL Offs(pOrigin,127.44,-106.79,-0.00),v40,z0,tcp\WObj:=Plywood;
    MoveL Offs(pOrigin,130.42,-107.71,-0.00),v40,z0,tcp\WObj:=Plywood;
    MoveL Offs(pOrigin,132.76,-109.12,-0.00),v40,z0,tcp\WObj:=Plywood;
    MoveL Offs(pOrigin,133.68,-110.12,-0.00),v40,z0,tcp\WObj:=Plywood;
    MoveL Offs(pOrigin,130.10,-107.92,-0.00),v40,z0,tcp\WObj:=Plywood;
    MoveL Offs(pOrigin,123.94,-106.68,-0.00),v40,fine,tcp\WObj:=Plywood;
    MoveL Offs(pOrigin,123.94,-106.68,-6.00),v60,z5,tcp\WObj:=Plywood;
    MoveL Offs(pOrigin,125.21,-103.07,-6.00),vTravel,z5,tcp\WObj:=Plywood;
    MoveL Offs(pOrigin,125.21,-103.07,-0.00),v60,z0,tcp\WObj:=Plywood;
    MoveL Offs(pOrigin,122.52,-101.90,-0.00),v40,z0,tcp\WObj:=Plywood;
    MoveL Offs(pOrigin,125.64,-102.96,-0.00),v40,z0,tcp\WObj:=Plywood;
    MoveL Offs(pOrigin,129.04,-102.64,-0.00),v40,z0,tcp\WObj:=Plywood;
    MoveL Offs(pOrigin,130.99,-102.96,-0.00),v40,z0,tcp\WObj:=Plywood;
    MoveL Offs(pOrigin,125.21,-103.07,-0.00),v40,fine,tcp\WObj:=Plywood;
    MoveL Offs(pOrigin,125.21,-103.07,-6.00),v60,z5,tcp\WObj:=Plywood;
    MoveL Offs(pOrigin,118.73,-93.51,-6.00),vTravel,z5,tcp\WObj:=Plywood;
    MoveL Offs(pOrigin,118.73,-93.51,-0.00),v60,z0,tcp\WObj:=Plywood;
    MoveL Offs(pOrigin,117.99,-93.68,-0.00),v40,z0,tcp\WObj:=Plywood;
    MoveL Offs(pOrigin,117.46,-92.87,-0.00),v40,z0,tcp\WObj:=Plywood;
    MoveL Offs(pOrigin,118.20,-91.17,-0.00),v40,z0,tcp\WObj:=Plywood;
    MoveL Offs(pOrigin,119.26,-90.89,-0.00),v40,z0,tcp\WObj:=Plywood;
    MoveL Offs(pOrigin,119.58,-91.38,-0.00),v40,z0,tcp\WObj:=Plywood;
    MoveL Offs(pOrigin,119.40,-92.55,-0.00),v40,z0,tcp\WObj:=Plywood;
    MoveL Offs(pOrigin,118.73,-93.51,-0.00),v40,z0,tcp\WObj:=Plywood;
    MoveL Offs(pOrigin,118.52,-93.40,-0.00),v40,z0,tcp\WObj:=Plywood;
    MoveL Offs(pOrigin,119.30,-92.34,-0.00),v40,z0,tcp\WObj:=Plywood;
    MoveL Offs(pOrigin,119.37,-91.38,-0.00),v40,z0,tcp\WObj:=Plywood;
    MoveL Offs(pOrigin,119.05,-90.99,-0.00),v40,z0,tcp\WObj:=Plywood;
    MoveL Offs(pOrigin,117.95,-91.70,-0.00),v40,z0,tcp\WObj:=Plywood;
    MoveL Offs(pOrigin,117.63,-92.76,-0.00),v40,z0,tcp\WObj:=Plywood;
    MoveL Offs(pOrigin,117.88,-93.47,-0.00),v40,z0,tcp\WObj:=Plywood;
    MoveL Offs(pOrigin,118.52,-93.40,-0.00),v40,fine,tcp\WObj:=Plywood;
    MoveL Offs(pOrigin,118.52,-93.40,-6.00),v60,z5,tcp\WObj:=Plywood;
    MoveL Offs(pOrigin,120.82,-85.15,-6.00),vTravel,z5,tcp\WObj:=Plywood;
    MoveL Offs(pOrigin,120.82,-85.15,-0.00),v60,z0,tcp\WObj:=Plywood;
    MoveL Offs(pOrigin,121.21,-84.55,-0.00),v40,z0,tcp\WObj:=Plywood;
    MoveL Offs(pOrigin,120.82,-85.15,-0.00),v40,fine,tcp\WObj:=Plywood;
    MoveL Offs(pOrigin,120.82,-85.15,-6.00),v60,z5,tcp\WObj:=Plywood;
    MoveL Offs(pOrigin,125.39,-79.69,-6.00),vTravel,z5,tcp\WObj:=Plywood;
    MoveL Offs(pOrigin,125.39,-79.69,-0.00),v60,z0,tcp\WObj:=Plywood;
    MoveL Offs(pOrigin,125.21,-78.53,-0.00),v40,z0,tcp\WObj:=Plywood;
    MoveL Offs(pOrigin,125.64,-77.82,-0.00),v40,z0,tcp\WObj:=Plywood;
    MoveL Offs(pOrigin,126.91,-77.36,-0.00),v40,z0,tcp\WObj:=Plywood;
    MoveL Offs(pOrigin,127.87,-77.99,-0.00),v40,z0,tcp\WObj:=Plywood;
    MoveL Offs(pOrigin,128.19,-79.16,-0.00),v40,z0,tcp\WObj:=Plywood;
    MoveL Offs(pOrigin,127.76,-80.01,-0.00),v40,z0,tcp\WObj:=Plywood;
    MoveL Offs(pOrigin,126.38,-80.44,-0.00),v40,z0,tcp\WObj:=Plywood;
    MoveL Offs(pOrigin,125.39,-79.69,-0.00),v40,z0,tcp\WObj:=Plywood;
    MoveL Offs(pOrigin,125.64,-79.69,-0.00),v40,z0,tcp\WObj:=Plywood;
    MoveL Offs(pOrigin,126.59,-80.30,-0.00),v40,z0,tcp\WObj:=Plywood;
    MoveL Offs(pOrigin,127.44,-80.01,-0.00),v40,z0,tcp\WObj:=Plywood;
    MoveL Offs(pOrigin,127.97,-79.16,-0.00),v40,z0,tcp\WObj:=Plywood;
    MoveL Offs(pOrigin,127.80,-78.21,-0.00),v40,z0,tcp\WObj:=Plywood;
    MoveL Offs(pOrigin,126.91,-77.57,-0.00),v40,z0,tcp\WObj:=Plywood;
    MoveL Offs(pOrigin,125.85,-77.89,-0.00),v40,z0,tcp\WObj:=Plywood;
    MoveL Offs(pOrigin,125.35,-78.84,-0.00),v40,z0,tcp\WObj:=Plywood;
    MoveL Offs(pOrigin,125.64,-79.69,-0.00),v40,fine,tcp\WObj:=Plywood;
    MoveL Offs(pOrigin,125.64,-79.69,-6.00),v60,z5,tcp\WObj:=Plywood;
    MoveL Offs(pOrigin,128.58,-83.80,-6.00),vTravel,z5,tcp\WObj:=Plywood;
    MoveL Offs(pOrigin,128.58,-83.80,-0.00),v60,z0,tcp\WObj:=Plywood;
    MoveL Offs(pOrigin,131.59,-86.07,-0.00),v40,z0,tcp\WObj:=Plywood;
    MoveL Offs(pOrigin,134.10,-89.40,-0.00),v40,z0,tcp\WObj:=Plywood;
    MoveL Offs(pOrigin,131.80,-86.60,-0.00),v40,z0,tcp\WObj:=Plywood;
    MoveL Offs(pOrigin,128.58,-83.80,-0.00),v40,fine,tcp\WObj:=Plywood;
    MoveL Offs(pOrigin,128.58,-83.80,-6.00),v60,z5,tcp\WObj:=Plywood;
    MoveL Offs(pOrigin,137.68,-90.67,-6.00),vTravel,z5,tcp\WObj:=Plywood;
    MoveL Offs(pOrigin,137.68,-90.67,-0.00),v60,z0,tcp\WObj:=Plywood;
    MoveL Offs(pOrigin,137.18,-89.96,-0.00),v40,z0,tcp\WObj:=Plywood;
    MoveL Offs(pOrigin,137.68,-90.67,-0.00),v40,fine,tcp\WObj:=Plywood;
    MoveL Offs(pOrigin,137.68,-90.67,-6.00),v60,z5,tcp\WObj:=Plywood;
    MoveL Offs(pOrigin,138.88,-91.63,-6.00),vTravel,z5,tcp\WObj:=Plywood;
    MoveL Offs(pOrigin,138.88,-91.63,-0.00),v60,z0,tcp\WObj:=Plywood;
    MoveL Offs(pOrigin,134.99,-82.85,-0.00),v40,z0,tcp\WObj:=Plywood;
    MoveL Offs(pOrigin,138.88,-91.63,-0.00),v40,fine,tcp\WObj:=Plywood;
    MoveL Offs(pOrigin,138.88,-91.63,-6.00),v60,z5,tcp\WObj:=Plywood;
    MoveL Offs(pOrigin,136.97,-110.15,-6.00),vTravel,z5,tcp\WObj:=Plywood;
    MoveL Offs(pOrigin,136.97,-110.15,-0.00),v60,z0,tcp\WObj:=Plywood;
    MoveL Offs(pOrigin,138.49,-111.14,-0.00),v40,z0,tcp\WObj:=Plywood;
    MoveL Offs(pOrigin,140.12,-112.99,-0.00),v40,z0,tcp\WObj:=Plywood;
    MoveL Offs(pOrigin,136.97,-110.15,-0.00),v40,fine,tcp\WObj:=Plywood;
    MoveL Offs(pOrigin,136.97,-110.15,-6.00),v60,z5,tcp\WObj:=Plywood;
    MoveL Offs(pOrigin,115.58,-125.63,-6.00),vTravel,z5,tcp\WObj:=Plywood;
  ENDPROC

  PROC DrawPart27()
    MoveL Offs(pOrigin,115.58,-125.63,-0.00),v60,z0,tcp\WObj:=Plywood;
    MoveL Offs(pOrigin,111.54,-119.50,-0.00),v40,z0,tcp\WObj:=Plywood;
    MoveL Offs(pOrigin,115.58,-125.63,-0.00),v40,fine,tcp\WObj:=Plywood;
    MoveL Offs(pOrigin,115.58,-125.63,-6.00),v60,z5,tcp\WObj:=Plywood;
    MoveL Offs(pOrigin,102.51,-122.34,-6.00),vTravel,z5,tcp\WObj:=Plywood;
    MoveL Offs(pOrigin,102.51,-122.34,-0.00),v60,z0,tcp\WObj:=Plywood;
    MoveL Offs(pOrigin,101.09,-125.70,-0.00),v40,z0,tcp\WObj:=Plywood;
    MoveL Offs(pOrigin,100.67,-129.14,-0.00),v40,z0,tcp\WObj:=Plywood;
    MoveL Offs(pOrigin,100.53,-126.76,-0.00),v40,z0,tcp\WObj:=Plywood;
    MoveL Offs(pOrigin,102.51,-122.34,-0.00),v40,fine,tcp\WObj:=Plywood;
    MoveL Offs(pOrigin,102.51,-122.34,-6.00),v60,z5,tcp\WObj:=Plywood;
    MoveL Offs(pOrigin,100.78,-121.84,-6.00),vTravel,z5,tcp\WObj:=Plywood;
    MoveL Offs(pOrigin,100.78,-121.84,-0.00),v60,z0,tcp\WObj:=Plywood;
    MoveL Offs(pOrigin,101.09,-119.54,-0.00),v40,z0,tcp\WObj:=Plywood;
    MoveL Offs(pOrigin,94.40,-117.66,-0.00),v40,z0,tcp\WObj:=Plywood;
    MoveL Offs(pOrigin,91.53,-116.28,-0.00),v40,z0,tcp\WObj:=Plywood;
    MoveL Offs(pOrigin,88.45,-113.80,-0.00),v40,z0,tcp\WObj:=Plywood;
    MoveL Offs(pOrigin,87.35,-112.21,-0.00),v40,z0,tcp\WObj:=Plywood;
    MoveL Offs(pOrigin,86.64,-110.26,-0.00),v40,z0,tcp\WObj:=Plywood;
    MoveL Offs(pOrigin,88.56,-113.48,-0.00),v40,z0,tcp\WObj:=Plywood;
    MoveL Offs(pOrigin,91.21,-115.64,-0.00),v40,z0,tcp\WObj:=Plywood;
    MoveL Offs(pOrigin,96.10,-117.77,-0.00),v40,z0,tcp\WObj:=Plywood;
    MoveL Offs(pOrigin,100.99,-118.90,-0.00),v40,z0,tcp\WObj:=Plywood;
    MoveL Offs(pOrigin,102.26,-116.46,-0.00),v40,z0,tcp\WObj:=Plywood;
    MoveL Offs(pOrigin,104.14,-115.93,-0.00),v40,z0,tcp\WObj:=Plywood;
    MoveL Offs(pOrigin,105.41,-112.95,-0.00),v40,z0,tcp\WObj:=Plywood;
    MoveL Offs(pOrigin,108.18,-109.44,-0.00),v40,z0,tcp\WObj:=Plywood;
    MoveL Offs(pOrigin,102.90,-108.59,-0.00),v40,z0,tcp\WObj:=Plywood;
    MoveL Offs(pOrigin,100.24,-107.78,-0.00),v40,z0,tcp\WObj:=Plywood;
    MoveL Offs(pOrigin,90.15,-102.82,-0.00),v40,z0,tcp\WObj:=Plywood;
    MoveL Offs(pOrigin,86.43,-101.40,-0.00),v40,z0,tcp\WObj:=Plywood;
    MoveL Offs(pOrigin,85.47,-104.03,-0.00),v40,z0,tcp\WObj:=Plywood;
    MoveL Offs(pOrigin,84.73,-108.28,-0.00),v40,z0,tcp\WObj:=Plywood;
    MoveL Offs(pOrigin,84.84,-111.57,-0.00),v40,z0,tcp\WObj:=Plywood;
    MoveL Offs(pOrigin,85.55,-114.22,-0.00),v40,z0,tcp\WObj:=Plywood;
    MoveL Offs(pOrigin,86.64,-116.14,-0.00),v40,z0,tcp\WObj:=Plywood;
    MoveL Offs(pOrigin,88.13,-117.52,-0.00),v40,z0,tcp\WObj:=Plywood;
    MoveL Offs(pOrigin,89.83,-118.51,-0.00),v40,z0,tcp\WObj:=Plywood;
    MoveL Offs(pOrigin,93.05,-119.68,-0.00),v40,z0,tcp\WObj:=Plywood;
    MoveL Offs(pOrigin,89.19,-118.83,-0.00),v40,z0,tcp\WObj:=Plywood;
    MoveL Offs(pOrigin,86.96,-117.52,-0.00),v40,z0,tcp\WObj:=Plywood;
    MoveL Offs(pOrigin,85.90,-116.35,-0.00),v40,z0,tcp\WObj:=Plywood;
    MoveL Offs(pOrigin,84.80,-114.33,-0.00),v40,z0,tcp\WObj:=Plywood;
    MoveL Offs(pOrigin,84.31,-112.53,-0.00),v40,z0,tcp\WObj:=Plywood;
    MoveL Offs(pOrigin,84.20,-107.21,-0.00),v40,z0,tcp\WObj:=Plywood;
    MoveL Offs(pOrigin,85.65,-101.16,-0.00),v40,z0,tcp\WObj:=Plywood;
    MoveL Offs(pOrigin,84.31,-100.55,-0.00),v40,z0,tcp\WObj:=Plywood;
    MoveL Offs(pOrigin,84.02,-100.73,-0.00),v40,z0,tcp\WObj:=Plywood;
    MoveL Offs(pOrigin,82.93,-106.68,-0.00),v40,z0,tcp\WObj:=Plywood;
    MoveL Offs(pOrigin,83.24,-112.31,-0.00),v40,z0,tcp\WObj:=Plywood;
    MoveL Offs(pOrigin,84.27,-115.29,-0.00),v40,z0,tcp\WObj:=Plywood;
    MoveL Offs(pOrigin,85.37,-117.06,-0.00),v40,z0,tcp\WObj:=Plywood;
    MoveL Offs(pOrigin,83.74,-115.07,-0.00),v40,z0,tcp\WObj:=Plywood;
    MoveL Offs(pOrigin,82.39,-111.14,-0.00),v40,z0,tcp\WObj:=Plywood;
    MoveL Offs(pOrigin,82.29,-106.36,-0.00),v40,z0,tcp\WObj:=Plywood;
    MoveL Offs(pOrigin,83.35,-100.41,-0.00),v40,z0,tcp\WObj:=Plywood;
    MoveL Offs(pOrigin,80.59,-99.56,-0.00),v40,z0,tcp\WObj:=Plywood;
    MoveL Offs(pOrigin,80.48,-104.56,-0.00),v40,z0,tcp\WObj:=Plywood;
    MoveL Offs(pOrigin,80.91,-110.51,-0.00),v40,z0,tcp\WObj:=Plywood;
    MoveL Offs(pOrigin,81.93,-113.80,-0.00),v40,z0,tcp\WObj:=Plywood;
    MoveL Offs(pOrigin,83.46,-116.03,-0.00),v40,z0,tcp\WObj:=Plywood;
    MoveL Offs(pOrigin,85.69,-117.87,-0.00),v40,z0,tcp\WObj:=Plywood;
    MoveL Offs(pOrigin,88.34,-119.15,-0.00),v40,z0,tcp\WObj:=Plywood;
    MoveL Offs(pOrigin,93.34,-120.60,-0.00),v40,z0,tcp\WObj:=Plywood;
    MoveL Offs(pOrigin,100.78,-121.84,-0.00),v40,fine,tcp\WObj:=Plywood;
    MoveL Offs(pOrigin,100.78,-121.84,-6.00),v60,z5,tcp\WObj:=Plywood;
    MoveL Offs(pOrigin,108.85,-108.70,-6.00),vTravel,z5,tcp\WObj:=Plywood;
    MoveL Offs(pOrigin,108.85,-108.70,-0.00),v60,z0,tcp\WObj:=Plywood;
    MoveL Offs(pOrigin,109.17,-108.70,-0.00),v40,z0,tcp\WObj:=Plywood;
    MoveL Offs(pOrigin,109.81,-107.85,-0.00),v40,z0,tcp\WObj:=Plywood;
    MoveL Offs(pOrigin,110.87,-100.52,-0.00),v40,z0,tcp\WObj:=Plywood;
    MoveL Offs(pOrigin,106.72,-96.91,-0.00),v40,z0,tcp\WObj:=Plywood;
    MoveL Offs(pOrigin,104.49,-95.42,-0.00),v40,z0,tcp\WObj:=Plywood;
    MoveL Offs(pOrigin,99.07,-97.33,-0.00),v40,z0,tcp\WObj:=Plywood;
    MoveL Offs(pOrigin,106.62,-106.36,-0.00),v40,z0,tcp\WObj:=Plywood;
    MoveL Offs(pOrigin,108.85,-108.70,-0.00),v40,fine,tcp\WObj:=Plywood;
    MoveL Offs(pOrigin,108.85,-108.70,-6.00),v60,z5,tcp\WObj:=Plywood;
    MoveL Offs(pOrigin,100.39,-101.72,-6.00),vTravel,z5,tcp\WObj:=Plywood;
    MoveL Offs(pOrigin,100.39,-101.72,-0.00),v60,z0,tcp\WObj:=Plywood;
    MoveL Offs(pOrigin,98.44,-100.09,-0.00),v40,z0,tcp\WObj:=Plywood;
    MoveL Offs(pOrigin,96.63,-97.97,-0.00),v40,z0,tcp\WObj:=Plywood;
    MoveL Offs(pOrigin,94.72,-94.14,-0.00),v40,z0,tcp\WObj:=Plywood;
    MoveL Offs(pOrigin,94.19,-91.28,-0.00),v40,z0,tcp\WObj:=Plywood;
    MoveL Offs(pOrigin,94.19,-87.88,-0.00),v40,z0,tcp\WObj:=Plywood;
    MoveL Offs(pOrigin,94.72,-83.70,-0.00),v40,z0,tcp\WObj:=Plywood;
    MoveL Offs(pOrigin,94.40,-90.11,-0.00),v40,z0,tcp\WObj:=Plywood;
    MoveL Offs(pOrigin,94.93,-93.82,-0.00),v40,z0,tcp\WObj:=Plywood;
    MoveL Offs(pOrigin,95.75,-96.06,-0.00),v40,z0,tcp\WObj:=Plywood;
    MoveL Offs(pOrigin,97.06,-98.18,-0.00),v40,z0,tcp\WObj:=Plywood;
    MoveL Offs(pOrigin,100.39,-101.72,-0.00),v40,fine,tcp\WObj:=Plywood;
    MoveL Offs(pOrigin,100.39,-101.72,-6.00),v60,z5,tcp\WObj:=Plywood;
    MoveL Offs(pOrigin,87.14,-88.97,-6.00),vTravel,z5,tcp\WObj:=Plywood;
    MoveL Offs(pOrigin,87.14,-88.97,-0.00),v60,z0,tcp\WObj:=Plywood;
    MoveL Offs(pOrigin,88.17,-87.13,-0.00),v40,z0,tcp\WObj:=Plywood;
    MoveL Offs(pOrigin,89.09,-84.37,-0.00),v40,z0,tcp\WObj:=Plywood;
    MoveL Offs(pOrigin,89.51,-80.44,-0.00),v40,z0,tcp\WObj:=Plywood;
    MoveL Offs(pOrigin,88.66,-74.17,-0.00),v40,z0,tcp\WObj:=Plywood;
    MoveL Offs(pOrigin,86.04,-67.23,-0.00),v40,z0,tcp\WObj:=Plywood;
    MoveL Offs(pOrigin,87.32,-69.49,-0.00),v40,z0,tcp\WObj:=Plywood;
    MoveL Offs(pOrigin,88.77,-73.32,-0.00),v40,z0,tcp\WObj:=Plywood;
    MoveL Offs(pOrigin,89.83,-78.95,-0.00),v40,z0,tcp\WObj:=Plywood;
    MoveL Offs(pOrigin,89.72,-82.56,-0.00),v40,z0,tcp\WObj:=Plywood;
    MoveL Offs(pOrigin,89.30,-84.69,-0.00),v40,z0,tcp\WObj:=Plywood;
    MoveL Offs(pOrigin,88.27,-87.34,-0.00),v40,z0,tcp\WObj:=Plywood;
    MoveL Offs(pOrigin,87.14,-88.97,-0.00),v40,fine,tcp\WObj:=Plywood;
    MoveL Offs(pOrigin,87.14,-88.97,-6.00),v60,z5,tcp\WObj:=Plywood;
    MoveL Offs(pOrigin,98.90,-61.24,-6.00),vTravel,z5,tcp\WObj:=Plywood;
    MoveL Offs(pOrigin,98.90,-61.24,-0.00),v60,z0,tcp\WObj:=Plywood;
    MoveL Offs(pOrigin,96.31,-59.29,-0.00),v40,z0,tcp\WObj:=Plywood;
    MoveL Offs(pOrigin,93.66,-56.53,-0.00),v40,z0,tcp\WObj:=Plywood;
    MoveL Offs(pOrigin,91.18,-53.03,-0.00),v40,z0,tcp\WObj:=Plywood;
    MoveL Offs(pOrigin,89.62,-49.91,-0.00),v40,z0,tcp\WObj:=Plywood;
    MoveL Offs(pOrigin,93.76,-56.21,-0.00),v40,z0,tcp\WObj:=Plywood;
    MoveL Offs(pOrigin,98.90,-61.24,-0.00),v40,fine,tcp\WObj:=Plywood;
    MoveL Offs(pOrigin,98.90,-61.24,-6.00),v60,z5,tcp\WObj:=Plywood;
    MoveL Offs(pOrigin,84.41,-50.58,-6.00),vTravel,z5,tcp\WObj:=Plywood;
    MoveL Offs(pOrigin,84.41,-50.58,-0.00),v60,z0,tcp\WObj:=Plywood;
    MoveL Offs(pOrigin,84.09,-49.84,-0.00),v40,z0,tcp\WObj:=Plywood;
    MoveL Offs(pOrigin,83.56,-49.45,-0.00),v40,z0,tcp\WObj:=Plywood;
    MoveL Offs(pOrigin,83.24,-49.62,-0.00),v40,z0,tcp\WObj:=Plywood;
  ENDPROC

  PROC DrawPart28()
    MoveL Offs(pOrigin,83.56,-50.58,-0.00),v40,z0,tcp\WObj:=Plywood;
    MoveL Offs(pOrigin,83.99,-50.79,-0.00),v40,z0,tcp\WObj:=Plywood;
    MoveL Offs(pOrigin,84.41,-50.58,-0.00),v40,fine,tcp\WObj:=Plywood;
    MoveL Offs(pOrigin,84.41,-50.58,-6.00),v60,z5,tcp\WObj:=Plywood;
    MoveL Offs(pOrigin,94.82,-26.32,-6.00),vTravel,z5,tcp\WObj:=Plywood;
    MoveL Offs(pOrigin,94.82,-26.32,-0.00),v60,z0,tcp\WObj:=Plywood;
    MoveL Offs(pOrigin,95.32,-26.04,-0.00),v40,z0,tcp\WObj:=Plywood;
    MoveL Offs(pOrigin,94.93,-25.01,-0.00),v40,z0,tcp\WObj:=Plywood;
    MoveL Offs(pOrigin,94.29,-25.29,-0.00),v40,z0,tcp\WObj:=Plywood;
    MoveL Offs(pOrigin,94.82,-26.32,-0.00),v40,z0,tcp\WObj:=Plywood;
    MoveL Offs(pOrigin,95.78,-26.00,-0.00),v40,z0,tcp\WObj:=Plywood;
    MoveL Offs(pOrigin,104.32,-23.49,-0.00),v40,z0,tcp\WObj:=Plywood;
    MoveL Offs(pOrigin,102.69,-21.86,-0.00),v40,z0,tcp\WObj:=Plywood;
    MoveL Offs(pOrigin,100.56,-21.04,-0.00),v40,z0,tcp\WObj:=Plywood;
    MoveL Offs(pOrigin,98.22,-20.83,-0.00),v40,z0,tcp\WObj:=Plywood;
    MoveL Offs(pOrigin,94.97,-21.58,-0.00),v40,z0,tcp\WObj:=Plywood;
    MoveL Offs(pOrigin,95.99,-23.38,-0.00),v40,z0,tcp\WObj:=Plywood;
    MoveL Offs(pOrigin,95.29,-24.87,-0.00),v40,z0,tcp\WObj:=Plywood;
    MoveL Offs(pOrigin,95.78,-26.00,-0.00),v40,fine,tcp\WObj:=Plywood;
    MoveL Offs(pOrigin,95.78,-26.00,-6.00),v60,z5,tcp\WObj:=Plywood;
    MoveL Offs(pOrigin,94.93,-24.66,-6.00),vTravel,z5,tcp\WObj:=Plywood;
    MoveL Offs(pOrigin,94.93,-24.66,-0.00),v60,z0,tcp\WObj:=Plywood;
    MoveL Offs(pOrigin,95.68,-23.38,-0.00),v40,z0,tcp\WObj:=Plywood;
    MoveL Offs(pOrigin,95.25,-22.32,-0.00),v40,z0,tcp\WObj:=Plywood;
    MoveL Offs(pOrigin,94.29,-21.79,-0.00),v40,z0,tcp\WObj:=Plywood;
    MoveL Offs(pOrigin,93.12,-22.11,-0.00),v40,z0,tcp\WObj:=Plywood;
    MoveL Offs(pOrigin,92.49,-23.27,-0.00),v40,z0,tcp\WObj:=Plywood;
    MoveL Offs(pOrigin,92.91,-24.34,-0.00),v40,z0,tcp\WObj:=Plywood;
    MoveL Offs(pOrigin,93.97,-24.94,-0.00),v40,z0,tcp\WObj:=Plywood;
    MoveL Offs(pOrigin,94.93,-24.66,-0.00),v40,z0,tcp\WObj:=Plywood;
    MoveL Offs(pOrigin,94.97,-24.20,-0.00),v40,z0,tcp\WObj:=Plywood;
    MoveL Offs(pOrigin,94.40,-24.55,-0.00),v40,z0,tcp\WObj:=Plywood;
    MoveL Offs(pOrigin,93.20,-24.20,-0.00),v40,z0,tcp\WObj:=Plywood;
    MoveL Offs(pOrigin,93.87,-24.55,-0.00),v40,z0,tcp\WObj:=Plywood;
    MoveL Offs(pOrigin,94.97,-24.20,-0.00),v40,fine,tcp\WObj:=Plywood;
    MoveL Offs(pOrigin,94.97,-24.20,-6.00),v60,z5,tcp\WObj:=Plywood;
    MoveL Offs(pOrigin,98.54,-13.61,-6.00),vTravel,z5,tcp\WObj:=Plywood;
    MoveL Offs(pOrigin,98.54,-13.61,-0.00),v60,z0,tcp\WObj:=Plywood;
    MoveL Offs(pOrigin,103.75,-13.15,-0.00),v40,z0,tcp\WObj:=Plywood;
    MoveL Offs(pOrigin,103.11,-11.27,-0.00),v40,z0,tcp\WObj:=Plywood;
    MoveL Offs(pOrigin,103.29,-9.89,-0.00),v40,z0,tcp\WObj:=Plywood;
    MoveL Offs(pOrigin,97.80,-10.38,-0.00),v40,z0,tcp\WObj:=Plywood;
    MoveL Offs(pOrigin,97.27,-11.27,-0.00),v40,z0,tcp\WObj:=Plywood;
    MoveL Offs(pOrigin,97.52,-12.76,-0.00),v40,z0,tcp\WObj:=Plywood;
    MoveL Offs(pOrigin,98.54,-13.61,-0.00),v40,z0,tcp\WObj:=Plywood;
    MoveL Offs(pOrigin,98.37,-12.83,-0.00),v40,z0,tcp\WObj:=Plywood;
    MoveL Offs(pOrigin,97.80,-11.69,-0.00),v40,z0,tcp\WObj:=Plywood;
    MoveL Offs(pOrigin,98.22,-10.74,-0.00),v40,z0,tcp\WObj:=Plywood;
    MoveL Offs(pOrigin,98.01,-12.01,-0.00),v40,z0,tcp\WObj:=Plywood;
    MoveL Offs(pOrigin,98.37,-12.83,-0.00),v40,fine,tcp\WObj:=Plywood;
    MoveL Offs(pOrigin,98.37,-12.83,-6.00),v60,z5,tcp\WObj:=Plywood;
    MoveL Offs(pOrigin,103.64,-11.06,-6.00),vTravel,z5,tcp\WObj:=Plywood;
    MoveL Offs(pOrigin,103.64,-11.06,-0.00),v60,z0,tcp\WObj:=Plywood;
    MoveL Offs(pOrigin,103.93,-12.12,-0.00),v40,z0,tcp\WObj:=Plywood;
    MoveL Offs(pOrigin,104.49,-12.69,-0.00),v40,z0,tcp\WObj:=Plywood;
    MoveL Offs(pOrigin,104.07,-11.38,-0.00),v40,z0,tcp\WObj:=Plywood;
    MoveL Offs(pOrigin,104.18,-9.75,-0.00),v40,z0,tcp\WObj:=Plywood;
    MoveL Offs(pOrigin,103.64,-11.06,-0.00),v40,fine,tcp\WObj:=Plywood;
    MoveL Offs(pOrigin,103.64,-11.06,-6.00),v60,z5,tcp\WObj:=Plywood;
    MoveL Offs(pOrigin,104.74,-10.52,-6.00),vTravel,z5,tcp\WObj:=Plywood;
    MoveL Offs(pOrigin,104.74,-10.52,-0.00),v60,z0,tcp\WObj:=Plywood;
    MoveL Offs(pOrigin,105.66,-10.84,-0.00),v40,z0,tcp\WObj:=Plywood;
    MoveL Offs(pOrigin,116.50,-9.78,-0.00),v40,z0,tcp\WObj:=Plywood;
    MoveL Offs(pOrigin,137.01,-15.09,-0.00),v40,z0,tcp\WObj:=Plywood;
    MoveL Offs(pOrigin,137.93,-14.56,-0.00),v40,z0,tcp\WObj:=Plywood;
    MoveL Offs(pOrigin,136.79,-14.03,-0.00),v40,z0,tcp\WObj:=Plywood;
    MoveL Offs(pOrigin,117.24,-8.93,-0.00),v40,z0,tcp\WObj:=Plywood;
    MoveL Offs(pOrigin,105.03,-10.06,-0.00),v40,z0,tcp\WObj:=Plywood;
    MoveL Offs(pOrigin,104.74,-10.52,-0.00),v40,z0,tcp\WObj:=Plywood;
    MoveL Offs(pOrigin,104.81,-11.48,-0.00),v40,z0,tcp\WObj:=Plywood;
    MoveL Offs(pOrigin,105.13,-12.23,-0.00),v40,z0,tcp\WObj:=Plywood;
    MoveL Offs(pOrigin,117.35,-11.27,-0.00),v40,z0,tcp\WObj:=Plywood;
    MoveL Offs(pOrigin,136.79,-16.05,-0.00),v40,z0,tcp\WObj:=Plywood;
    MoveL Offs(pOrigin,137.08,-15.62,-0.00),v40,z0,tcp\WObj:=Plywood;
    MoveL Offs(pOrigin,136.37,-15.20,-0.00),v40,z0,tcp\WObj:=Plywood;
    MoveL Offs(pOrigin,116.61,-10.14,-0.00),v40,z0,tcp\WObj:=Plywood;
    MoveL Offs(pOrigin,105.66,-11.16,-0.00),v40,z0,tcp\WObj:=Plywood;
    MoveL Offs(pOrigin,104.81,-11.48,-0.00),v40,fine,tcp\WObj:=Plywood;
    MoveL Offs(pOrigin,104.81,-11.48,-6.00),v60,z5,tcp\WObj:=Plywood;
    MoveL Offs(pOrigin,106.37,-12.76,-6.00),vTravel,z5,tcp\WObj:=Plywood;
    MoveL Offs(pOrigin,106.37,-12.76,-0.00),v60,z0,tcp\WObj:=Plywood;
    MoveL Offs(pOrigin,126.91,-17.33,-0.00),v40,z0,tcp\WObj:=Plywood;
    MoveL Offs(pOrigin,129.57,-16.37,-0.00),v40,z0,tcp\WObj:=Plywood;
    MoveL Offs(pOrigin,132.01,-16.37,-0.00),v40,z0,tcp\WObj:=Plywood;
    MoveL Offs(pOrigin,135.20,-16.90,-0.00),v40,z0,tcp\WObj:=Plywood;
    MoveL Offs(pOrigin,136.51,-16.69,-0.00),v40,z0,tcp\WObj:=Plywood;
    MoveL Offs(pOrigin,117.14,-11.69,-0.00),v40,z0,tcp\WObj:=Plywood;
    MoveL Offs(pOrigin,106.37,-12.76,-0.00),v40,fine,tcp\WObj:=Plywood;
    MoveL Offs(pOrigin,106.37,-12.76,-6.00),v60,z5,tcp\WObj:=Plywood;
    MoveL Offs(pOrigin,107.04,-23.63,-6.00),vTravel,z5,tcp\WObj:=Plywood;
    MoveL Offs(pOrigin,107.04,-23.63,-0.00),v60,z0,tcp\WObj:=Plywood;
    MoveL Offs(pOrigin,108.32,-25.79,-0.00),v40,z0,tcp\WObj:=Plywood;
    MoveL Offs(pOrigin,109.24,-25.19,-0.00),v40,z0,tcp\WObj:=Plywood;
    MoveL Offs(pOrigin,108.64,-23.52,-0.00),v40,z0,tcp\WObj:=Plywood;
    MoveL Offs(pOrigin,107.04,-23.63,-0.00),v40,fine,tcp\WObj:=Plywood;
    MoveL Offs(pOrigin,107.04,-23.63,-6.00),v60,z5,tcp\WObj:=Plywood;
    MoveL Offs(pOrigin,109.52,-23.70,-6.00),vTravel,z5,tcp\WObj:=Plywood;
    MoveL Offs(pOrigin,109.52,-23.70,-0.00),v60,z0,tcp\WObj:=Plywood;
    MoveL Offs(pOrigin,110.12,-24.69,-0.00),v40,z0,tcp\WObj:=Plywood;
    MoveL Offs(pOrigin,112.82,-23.27,-0.00),v40,z0,tcp\WObj:=Plywood;
    MoveL Offs(pOrigin,109.81,-23.38,-0.00),v40,z0,tcp\WObj:=Plywood;
    MoveL Offs(pOrigin,109.52,-23.70,-0.00),v40,fine,tcp\WObj:=Plywood;
    MoveL Offs(pOrigin,109.52,-23.70,-6.00),v60,z5,tcp\WObj:=Plywood;
    MoveL Offs(pOrigin,111.51,-24.51,-6.00),vTravel,z5,tcp\WObj:=Plywood;
    MoveL Offs(pOrigin,111.51,-24.51,-0.00),v60,z0,tcp\WObj:=Plywood;
    MoveL Offs(pOrigin,108.96,-26.14,-0.00),v40,z0,tcp\WObj:=Plywood;
    MoveL Offs(pOrigin,107.15,-28.38,-0.00),v40,z0,tcp\WObj:=Plywood;
    MoveL Offs(pOrigin,108.11,-28.66,-0.00),v40,z0,tcp\WObj:=Plywood;
    MoveL Offs(pOrigin,110.62,-26.32,-0.00),v40,z0,tcp\WObj:=Plywood;
    MoveL Offs(pOrigin,108.32,-28.59,-0.00),v40,z0,tcp\WObj:=Plywood;
    MoveL Offs(pOrigin,108.32,-28.91,-0.00),v40,z0,tcp\WObj:=Plywood;
    MoveL Offs(pOrigin,108.64,-28.91,-0.00),v40,z0,tcp\WObj:=Plywood;
    MoveL Offs(pOrigin,111.19,-26.14,-0.00),v40,z0,tcp\WObj:=Plywood;
    MoveL Offs(pOrigin,112.11,-24.66,-0.00),v40,z0,tcp\WObj:=Plywood;
    MoveL Offs(pOrigin,111.51,-24.51,-0.00),v40,z0,tcp\WObj:=Plywood;
    MoveL Offs(pOrigin,112.07,-24.44,-0.00),v40,z0,tcp\WObj:=Plywood;
    MoveL Offs(pOrigin,112.46,-24.44,-0.00),v40,z0,tcp\WObj:=Plywood;
    MoveL Offs(pOrigin,112.75,-23.91,-0.00),v40,z0,tcp\WObj:=Plywood;
    MoveL Offs(pOrigin,112.07,-24.44,-0.00),v40,fine,tcp\WObj:=Plywood;
    MoveL Offs(pOrigin,112.07,-24.44,-6.00),v60,z5,tcp\WObj:=Plywood;
  ENDPROC

  PROC DrawPart29()
    MoveL Offs(pOrigin,121.46,-22.00,-6.00),vTravel,z5,tcp\WObj:=Plywood;
    MoveL Offs(pOrigin,121.46,-22.00,-0.00),v60,z0,tcp\WObj:=Plywood;
    MoveL Offs(pOrigin,125.53,-27.10,-0.00),v40,z0,tcp\WObj:=Plywood;
    MoveL Offs(pOrigin,129.99,-31.24,-0.00),v40,z0,tcp\WObj:=Plywood;
    MoveL Offs(pOrigin,132.44,-32.55,-0.00),v40,z0,tcp\WObj:=Plywood;
    MoveL Offs(pOrigin,133.50,-32.52,-0.00),v40,z0,tcp\WObj:=Plywood;
    MoveL Offs(pOrigin,134.70,-30.92,-0.00),v40,z0,tcp\WObj:=Plywood;
    MoveL Offs(pOrigin,134.99,-29.65,-0.00),v40,z0,tcp\WObj:=Plywood;
    MoveL Offs(pOrigin,131.91,-28.20,-0.00),v40,z0,tcp\WObj:=Plywood;
    MoveL Offs(pOrigin,124.08,-22.50,-0.00),v40,z0,tcp\WObj:=Plywood;
    MoveL Offs(pOrigin,121.92,-20.19,-0.00),v40,z0,tcp\WObj:=Plywood;
    MoveL Offs(pOrigin,121.28,-21.26,-0.00),v40,z0,tcp\WObj:=Plywood;
    MoveL Offs(pOrigin,121.46,-22.00,-0.00),v40,fine,tcp\WObj:=Plywood;
    MoveL Offs(pOrigin,121.46,-22.00,-6.00),v60,z5,tcp\WObj:=Plywood;
    MoveL Offs(pOrigin,126.03,-17.64,-6.00),vTravel,z5,tcp\WObj:=Plywood;
    MoveL Offs(pOrigin,126.03,-17.64,-0.00),v60,z0,tcp\WObj:=Plywood;
    MoveL Offs(pOrigin,126.98,-17.96,-0.00),v40,z0,tcp\WObj:=Plywood;
    MoveL Offs(pOrigin,126.81,-17.64,-0.00),v40,z0,tcp\WObj:=Plywood;
    MoveL Offs(pOrigin,126.03,-17.64,-0.00),v40,fine,tcp\WObj:=Plywood;
    MoveL Offs(pOrigin,126.03,-17.64,-6.00),v60,z5,tcp\WObj:=Plywood;
    MoveL Offs(pOrigin,127.66,-18.07,-6.00),vTravel,z5,tcp\WObj:=Plywood;
    MoveL Offs(pOrigin,127.66,-18.07,-0.00),v60,z0,tcp\WObj:=Plywood;
    MoveL Offs(pOrigin,127.97,-18.92,-0.00),v40,z0,tcp\WObj:=Plywood;
    MoveL Offs(pOrigin,129.89,-20.23,-0.00),v40,z0,tcp\WObj:=Plywood;
    MoveL Offs(pOrigin,139.98,-24.98,-0.00),v40,z0,tcp\WObj:=Plywood;
    MoveL Offs(pOrigin,140.83,-25.12,-0.00),v40,z0,tcp\WObj:=Plywood;
    MoveL Offs(pOrigin,141.57,-24.76,-0.00),v40,z0,tcp\WObj:=Plywood;
    MoveL Offs(pOrigin,142.74,-21.89,-0.00),v40,z0,tcp\WObj:=Plywood;
    MoveL Offs(pOrigin,142.85,-20.62,-0.00),v40,z0,tcp\WObj:=Plywood;
    MoveL Offs(pOrigin,142.32,-20.05,-0.00),v40,z0,tcp\WObj:=Plywood;
    MoveL Offs(pOrigin,135.31,-17.54,-0.00),v40,z0,tcp\WObj:=Plywood;
    MoveL Offs(pOrigin,131.80,-16.90,-0.00),v40,z0,tcp\WObj:=Plywood;
    MoveL Offs(pOrigin,129.89,-16.90,-0.00),v40,z0,tcp\WObj:=Plywood;
    MoveL Offs(pOrigin,128.40,-17.18,-0.00),v40,z0,tcp\WObj:=Plywood;
    MoveL Offs(pOrigin,127.66,-18.07,-0.00),v40,fine,tcp\WObj:=Plywood;
    MoveL Offs(pOrigin,127.66,-18.07,-6.00),v60,z5,tcp\WObj:=Plywood;
    MoveL Offs(pOrigin,135.59,-30.08,-6.00),vTravel,z5,tcp\WObj:=Plywood;
    MoveL Offs(pOrigin,135.59,-30.08,-0.00),v60,z0,tcp\WObj:=Plywood;
    MoveL Offs(pOrigin,133.61,-33.12,-0.00),v40,z0,tcp\WObj:=Plywood;
    MoveL Offs(pOrigin,134.92,-31.77,-0.00),v40,z0,tcp\WObj:=Plywood;
    MoveL Offs(pOrigin,135.59,-30.08,-0.00),v40,z0,tcp\WObj:=Plywood;
    MoveL Offs(pOrigin,135.84,-30.08,-0.00),v40,z0,tcp\WObj:=Plywood;
    MoveL Offs(pOrigin,134.03,-33.33,-0.00),v40,z0,tcp\WObj:=Plywood;
    MoveL Offs(pOrigin,134.88,-33.51,-0.00),v40,z0,tcp\WObj:=Plywood;
    MoveL Offs(pOrigin,135.73,-32.73,-0.00),v40,z0,tcp\WObj:=Plywood;
    MoveL Offs(pOrigin,136.76,-30.39,-0.00),v40,z0,tcp\WObj:=Plywood;
    MoveL Offs(pOrigin,135.52,-32.62,-0.00),v40,z0,tcp\WObj:=Plywood;
    MoveL Offs(pOrigin,134.74,-33.23,-0.00),v40,z0,tcp\WObj:=Plywood;
    MoveL Offs(pOrigin,136.40,-30.50,-0.00),v40,z0,tcp\WObj:=Plywood;
    MoveL Offs(pOrigin,135.84,-30.08,-0.00),v40,fine,tcp\WObj:=Plywood;
    MoveL Offs(pOrigin,135.84,-30.08,-6.00),v60,z5,tcp\WObj:=Plywood;
    MoveL Offs(pOrigin,141.40,-25.29,-6.00),vTravel,z5,tcp\WObj:=Plywood;
    MoveL Offs(pOrigin,141.40,-25.29,-0.00),v60,z0,tcp\WObj:=Plywood;
    MoveL Offs(pOrigin,142.43,-25.83,-0.00),v40,z0,tcp\WObj:=Plywood;
    MoveL Offs(pOrigin,143.42,-25.61,-0.00),v40,z0,tcp\WObj:=Plywood;
    MoveL Offs(pOrigin,141.89,-24.98,-0.00),v40,z0,tcp\WObj:=Plywood;
    MoveL Offs(pOrigin,141.40,-25.29,-0.00),v40,z0,tcp\WObj:=Plywood;
    MoveL Offs(pOrigin,142.11,-24.66,-0.00),v40,z0,tcp\WObj:=Plywood;
    MoveL Offs(pOrigin,144.23,-25.51,-0.00),v40,z0,tcp\WObj:=Plywood;
    MoveL Offs(pOrigin,144.90,-24.76,-0.00),v40,z0,tcp\WObj:=Plywood;
    MoveL Offs(pOrigin,145.72,-22.00,-0.00),v40,z0,tcp\WObj:=Plywood;
    MoveL Offs(pOrigin,145.40,-21.61,-0.00),v40,z0,tcp\WObj:=Plywood;
    MoveL Offs(pOrigin,143.49,-20.94,-0.00),v40,z0,tcp\WObj:=Plywood;
    MoveL Offs(pOrigin,142.11,-24.66,-0.00),v40,z0,tcp\WObj:=Plywood;
    MoveL Offs(pOrigin,142.71,-24.23,-0.00),v40,z0,tcp\WObj:=Plywood;
    MoveL Offs(pOrigin,143.66,-21.75,-0.00),v40,z0,tcp\WObj:=Plywood;
    MoveL Offs(pOrigin,142.85,-24.23,-0.00),v40,z0,tcp\WObj:=Plywood;
    MoveL Offs(pOrigin,144.30,-24.94,-0.00),v40,z0,tcp\WObj:=Plywood;
    MoveL Offs(pOrigin,142.71,-24.23,-0.00),v40,z0,tcp\WObj:=Plywood;
    MoveL Offs(pOrigin,143.42,-23.77,-0.00),v40,z0,tcp\WObj:=Plywood;
    MoveL Offs(pOrigin,143.88,-23.20,-0.00),v40,z0,tcp\WObj:=Plywood;
    MoveL Offs(pOrigin,143.42,-23.77,-0.00),v40,z0,tcp\WObj:=Plywood;
    MoveL Offs(pOrigin,144.02,-23.70,-0.00),v40,z0,tcp\WObj:=Plywood;
    MoveL Offs(pOrigin,144.44,-23.49,-0.00),v40,z0,tcp\WObj:=Plywood;
    MoveL Offs(pOrigin,144.44,-23.81,-0.00),v40,z0,tcp\WObj:=Plywood;
    MoveL Offs(pOrigin,144.02,-23.70,-0.00),v40,z0,tcp\WObj:=Plywood;
    MoveL Offs(pOrigin,144.44,-23.49,-0.00),v40,z0,tcp\WObj:=Plywood;
    MoveL Offs(pOrigin,144.44,-23.81,-0.00),v40,z0,tcp\WObj:=Plywood;
    MoveL Offs(pOrigin,144.02,-23.70,-0.00),v40,z0,tcp\WObj:=Plywood;
    MoveL Offs(pOrigin,144.94,-23.45,-0.00),v40,z0,tcp\WObj:=Plywood;
    MoveL Offs(pOrigin,145.05,-22.21,-0.00),v40,z0,tcp\WObj:=Plywood;
    MoveL Offs(pOrigin,144.16,-21.82,-0.00),v40,z0,tcp\WObj:=Plywood;
    MoveL Offs(pOrigin,145.19,-22.32,-0.00),v40,z0,tcp\WObj:=Plywood;
    MoveL Offs(pOrigin,144.94,-23.45,-0.00),v40,fine,tcp\WObj:=Plywood;
    MoveL Offs(pOrigin,144.94,-23.45,-6.00),v60,z5,tcp\WObj:=Plywood;
    MoveL Offs(pOrigin,143.84,-22.71,-6.00),vTravel,z5,tcp\WObj:=Plywood;
    MoveL Offs(pOrigin,143.84,-22.71,-0.00),v60,z0,tcp\WObj:=Plywood;
    MoveL Offs(pOrigin,144.09,-22.25,-0.00),v40,z0,tcp\WObj:=Plywood;
    MoveL Offs(pOrigin,143.84,-22.71,-0.00),v40,fine,tcp\WObj:=Plywood;
    MoveL Offs(pOrigin,143.84,-22.71,-6.00),v60,z5,tcp\WObj:=Plywood;
    MoveL Offs(pOrigin,143.20,-20.51,-6.00),vTravel,z5,tcp\WObj:=Plywood;
    MoveL Offs(pOrigin,143.20,-20.51,-0.00),v60,z0,tcp\WObj:=Plywood;
    MoveL Offs(pOrigin,143.74,-20.62,-0.00),v40,z0,tcp\WObj:=Plywood;
    MoveL Offs(pOrigin,143.20,-20.51,-0.00),v40,fine,tcp\WObj:=Plywood;
    MoveL Offs(pOrigin,143.20,-20.51,-6.00),v60,z5,tcp\WObj:=Plywood;
    MoveL Offs(pOrigin,157.48,-18.53,-6.00),vTravel,z5,tcp\WObj:=Plywood;
    MoveL Offs(pOrigin,157.48,-18.53,-0.00),v60,z0,tcp\WObj:=Plywood;
    MoveL Offs(pOrigin,156.59,-17.40,-0.00),v40,z0,tcp\WObj:=Plywood;
    MoveL Offs(pOrigin,157.48,-18.53,-0.00),v40,fine,tcp\WObj:=Plywood;
    MoveL Offs(pOrigin,157.48,-18.53,-6.00),v60,z5,tcp\WObj:=Plywood;
    MoveL Offs(pOrigin,157.48,-16.58,-6.00),vTravel,z5,tcp\WObj:=Plywood;
    MoveL Offs(pOrigin,157.48,-16.58,-0.00),v60,z0,tcp\WObj:=Plywood;
    MoveL Offs(pOrigin,160.66,-18.07,-0.00),v40,z0,tcp\WObj:=Plywood;
    MoveL Offs(pOrigin,160.27,-17.22,-0.00),v40,z0,tcp\WObj:=Plywood;
    MoveL Offs(pOrigin,159.32,-16.55,-0.00),v40,z0,tcp\WObj:=Plywood;
    MoveL Offs(pOrigin,157.48,-16.58,-0.00),v40,fine,tcp\WObj:=Plywood;
    MoveL Offs(pOrigin,157.48,-16.58,-6.00),v60,z5,tcp\WObj:=Plywood;
    MoveL Offs(pOrigin,168.07,-16.05,-6.00),vTravel,z5,tcp\WObj:=Plywood;
    MoveL Offs(pOrigin,168.07,-16.05,-0.00),v60,z0,tcp\WObj:=Plywood;
    MoveL Offs(pOrigin,170.69,-16.16,-0.00),v40,z0,tcp\WObj:=Plywood;
    MoveL Offs(pOrigin,171.96,-16.79,-0.00),v40,z0,tcp\WObj:=Plywood;
    MoveL Offs(pOrigin,173.27,-18.49,-0.00),v40,z0,tcp\WObj:=Plywood;
    MoveL Offs(pOrigin,174.44,-22.21,-0.00),v40,z0,tcp\WObj:=Plywood;
    MoveL Offs(pOrigin,174.69,-22.21,-0.00),v40,z0,tcp\WObj:=Plywood;
    MoveL Offs(pOrigin,174.73,-19.45,-0.00),v40,z0,tcp\WObj:=Plywood;
    MoveL Offs(pOrigin,173.91,-17.54,-0.00),v40,z0,tcp\WObj:=Plywood;
    MoveL Offs(pOrigin,172.71,-16.16,-0.00),v40,z0,tcp\WObj:=Plywood;
    MoveL Offs(pOrigin,170.90,-15.31,-0.00),v40,z0,tcp\WObj:=Plywood;
    MoveL Offs(pOrigin,169.20,-15.52,-0.00),v40,z0,tcp\WObj:=Plywood;
    MoveL Offs(pOrigin,168.07,-16.05,-0.00),v40,fine,tcp\WObj:=Plywood;
  ENDPROC

  PROC DrawPart30()
    MoveL Offs(pOrigin,168.07,-16.05,-6.00),v60,z5,tcp\WObj:=Plywood;
    MoveL Offs(pOrigin,170.23,-16.79,-6.00),vTravel,z5,tcp\WObj:=Plywood;
    MoveL Offs(pOrigin,170.23,-16.79,-0.00),v60,z0,tcp\WObj:=Plywood;
    MoveL Offs(pOrigin,171.47,-17.22,-0.00),v40,z0,tcp\WObj:=Plywood;
    MoveL Offs(pOrigin,170.90,-16.76,-0.00),v40,z0,tcp\WObj:=Plywood;
    MoveL Offs(pOrigin,170.23,-16.79,-0.00),v40,fine,tcp\WObj:=Plywood;
    MoveL Offs(pOrigin,170.23,-16.79,-6.00),v60,z5,tcp\WObj:=Plywood;
    MoveL Offs(pOrigin,170.16,-18.88,-6.00),vTravel,z5,tcp\WObj:=Plywood;
    MoveL Offs(pOrigin,170.16,-18.88,-0.00),v60,z0,tcp\WObj:=Plywood;
    MoveL Offs(pOrigin,171.15,-19.77,-0.00),v40,z0,tcp\WObj:=Plywood;
    MoveL Offs(pOrigin,171.32,-21.04,-0.00),v40,z0,tcp\WObj:=Plywood;
    MoveL Offs(pOrigin,170.58,-21.93,-0.00),v40,z0,tcp\WObj:=Plywood;
    MoveL Offs(pOrigin,169.62,-21.86,-0.00),v40,z0,tcp\WObj:=Plywood;
    MoveL Offs(pOrigin,168.81,-21.04,-0.00),v40,z0,tcp\WObj:=Plywood;
    MoveL Offs(pOrigin,168.56,-19.77,-0.00),v40,z0,tcp\WObj:=Plywood;
    MoveL Offs(pOrigin,169.20,-18.88,-0.00),v40,z0,tcp\WObj:=Plywood;
    MoveL Offs(pOrigin,170.16,-18.88,-0.00),v40,z0,tcp\WObj:=Plywood;
    MoveL Offs(pOrigin,170.16,-19.06,-0.00),v40,z0,tcp\WObj:=Plywood;
    MoveL Offs(pOrigin,169.31,-19.10,-0.00),v40,z0,tcp\WObj:=Plywood;
    MoveL Offs(pOrigin,168.67,-19.88,-0.00),v40,z0,tcp\WObj:=Plywood;
    MoveL Offs(pOrigin,168.85,-20.73,-0.00),v40,z0,tcp\WObj:=Plywood;
    MoveL Offs(pOrigin,169.31,-21.43,-0.00),v40,z0,tcp\WObj:=Plywood;
    MoveL Offs(pOrigin,170.37,-21.79,-0.00),v40,z0,tcp\WObj:=Plywood;
    MoveL Offs(pOrigin,171.15,-21.15,-0.00),v40,z0,tcp\WObj:=Plywood;
    MoveL Offs(pOrigin,171.15,-20.19,-0.00),v40,z0,tcp\WObj:=Plywood;
    MoveL Offs(pOrigin,170.16,-19.06,-0.00),v40,fine,tcp\WObj:=Plywood;
    MoveL Offs(pOrigin,170.16,-19.06,-6.00),v60,z5,tcp\WObj:=Plywood;
    MoveL Offs(pOrigin,169.55,-21.19,-6.00),vTravel,z5,tcp\WObj:=Plywood;
    MoveL Offs(pOrigin,169.55,-21.19,-0.00),v60,z0,tcp\WObj:=Plywood;
    MoveL Offs(pOrigin,169.09,-20.26,-0.00),v40,z0,tcp\WObj:=Plywood;
    MoveL Offs(pOrigin,169.55,-21.19,-0.00),v40,fine,tcp\WObj:=Plywood;
    MoveL Offs(pOrigin,169.55,-21.19,-6.00),v60,z5,tcp\WObj:=Plywood;
    MoveL Offs(pOrigin,177.27,-22.14,-6.00),vTravel,z5,tcp\WObj:=Plywood;
    MoveL Offs(pOrigin,177.27,-22.14,-0.00),v60,z0,tcp\WObj:=Plywood;
    MoveL Offs(pOrigin,176.43,-19.31,-0.00),v40,z0,tcp\WObj:=Plywood;
    MoveL Offs(pOrigin,177.27,-22.14,-0.00),v40,fine,tcp\WObj:=Plywood;
    MoveL Offs(pOrigin,177.27,-22.14,-6.00),v60,z5,tcp\WObj:=Plywood;
    MoveL Offs(pOrigin,185.85,-31.39,-6.00),vTravel,z5,tcp\WObj:=Plywood;
    MoveL Offs(pOrigin,185.85,-31.39,-0.00),v60,z0,tcp\WObj:=Plywood;
    MoveL Offs(pOrigin,193.07,-24.73,-0.00),v40,z0,tcp\WObj:=Plywood;
    MoveL Offs(pOrigin,188.96,-28.91,-0.00),v40,z0,tcp\WObj:=Plywood;
    MoveL Offs(pOrigin,185.85,-31.39,-0.00),v40,fine,tcp\WObj:=Plywood;
    MoveL Offs(pOrigin,185.85,-31.39,-6.00),v60,z5,tcp\WObj:=Plywood;
    MoveL Offs(pOrigin,202.28,-37.97,-6.00),vTravel,z5,tcp\WObj:=Plywood;
    MoveL Offs(pOrigin,202.28,-37.97,-0.00),v60,z0,tcp\WObj:=Plywood;
    MoveL Offs(pOrigin,203.55,-36.20,-0.00),v40,z0,tcp\WObj:=Plywood;
    MoveL Offs(pOrigin,202.28,-37.97,-0.00),v40,fine,tcp\WObj:=Plywood;
    MoveL Offs(pOrigin,202.28,-37.97,-6.00),v60,z5,tcp\WObj:=Plywood;
    MoveL Offs(pOrigin,127.12,-59.19,-6.00),vTravel,z5,tcp\WObj:=Plywood;
    MoveL Offs(pOrigin,127.12,-59.19,-0.00),v60,z0,tcp\WObj:=Plywood;
    MoveL Offs(pOrigin,126.59,-60.25,-0.00),v40,z0,tcp\WObj:=Plywood;
    MoveL Offs(pOrigin,125.53,-60.67,-0.00),v40,z0,tcp\WObj:=Plywood;
    MoveL Offs(pOrigin,124.36,-60.04,-0.00),v40,z0,tcp\WObj:=Plywood;
    MoveL Offs(pOrigin,124.04,-58.76,-0.00),v40,z0,tcp\WObj:=Plywood;
    MoveL Offs(pOrigin,124.79,-57.77,-0.00),v40,z0,tcp\WObj:=Plywood;
    MoveL Offs(pOrigin,125.96,-57.59,-0.00),v40,z0,tcp\WObj:=Plywood;
    MoveL Offs(pOrigin,126.70,-58.02,-0.00),v40,z0,tcp\WObj:=Plywood;
    MoveL Offs(pOrigin,127.12,-59.19,-0.00),v40,z0,tcp\WObj:=Plywood;
    MoveL Offs(pOrigin,126.91,-59.29,-0.00),v40,z0,tcp\WObj:=Plywood;
    MoveL Offs(pOrigin,126.59,-58.23,-0.00),v40,z0,tcp\WObj:=Plywood;
    MoveL Offs(pOrigin,125.64,-57.70,-0.00),v40,z0,tcp\WObj:=Plywood;
    MoveL Offs(pOrigin,124.57,-58.12,-0.00),v40,z0,tcp\WObj:=Plywood;
    MoveL Offs(pOrigin,124.26,-58.76,-0.00),v40,z0,tcp\WObj:=Plywood;
    MoveL Offs(pOrigin,124.57,-60.04,-0.00),v40,z0,tcp\WObj:=Plywood;
    MoveL Offs(pOrigin,125.43,-60.46,-0.00),v40,z0,tcp\WObj:=Plywood;
    MoveL Offs(pOrigin,126.28,-60.25,-0.00),v40,z0,tcp\WObj:=Plywood;
    MoveL Offs(pOrigin,126.91,-59.29,-0.00),v40,fine,tcp\WObj:=Plywood;
    MoveL Offs(pOrigin,126.91,-59.29,-6.00),v60,z5,tcp\WObj:=Plywood;
    MoveL Offs(pOrigin,117.78,-70.27,-6.00),vTravel,z5,tcp\WObj:=Plywood;
    MoveL Offs(pOrigin,117.78,-70.27,-0.00),v60,z0,tcp\WObj:=Plywood;
    MoveL Offs(pOrigin,118.62,-66.38,-0.00),v40,z0,tcp\WObj:=Plywood;
    MoveL Offs(pOrigin,117.78,-70.27,-0.00),v40,fine,tcp\WObj:=Plywood;
    MoveL Offs(pOrigin,117.78,-70.27,-6.00),v60,z5,tcp\WObj:=Plywood;
    MoveL Offs(pOrigin,138.18,-137.32,-6.00),vTravel,z5,tcp\WObj:=Plywood;
    MoveL Offs(pOrigin,138.18,-137.32,-0.00),v60,z0,tcp\WObj:=Plywood;
    MoveL Offs(pOrigin,137.86,-138.77,-0.00),v40,z0,tcp\WObj:=Plywood;
    MoveL Offs(pOrigin,139.56,-138.88,-0.00),v40,z0,tcp\WObj:=Plywood;
    MoveL Offs(pOrigin,139.56,-138.45,-0.00),v40,z0,tcp\WObj:=Plywood;
    MoveL Offs(pOrigin,138.67,-138.06,-0.00),v40,z0,tcp\WObj:=Plywood;
    MoveL Offs(pOrigin,139.45,-138.24,-0.00),v40,z0,tcp\WObj:=Plywood;
    MoveL Offs(pOrigin,139.56,-137.92,-0.00),v40,z0,tcp\WObj:=Plywood;
    MoveL Offs(pOrigin,138.18,-137.32,-0.00),v40,fine,tcp\WObj:=Plywood;
    MoveL Offs(pOrigin,138.18,-137.32,-6.00),v60,z5,tcp\WObj:=Plywood;
    MoveL Offs(pOrigin,140.30,-138.45,-6.00),vTravel,z5,tcp\WObj:=Plywood;
    MoveL Offs(pOrigin,140.30,-138.45,-0.00),v60,z0,tcp\WObj:=Plywood;
    MoveL Offs(pOrigin,142.14,-138.56,-0.00),v40,z0,tcp\WObj:=Plywood;
    MoveL Offs(pOrigin,140.30,-138.45,-0.00),v40,fine,tcp\WObj:=Plywood;
    MoveL Offs(pOrigin,140.30,-138.45,-6.00),v60,z5,tcp\WObj:=Plywood;
    MoveL Offs(pOrigin,141.68,-141.53,-6.00),vTravel,z5,tcp\WObj:=Plywood;
    MoveL Offs(pOrigin,141.68,-141.53,-0.00),v60,z0,tcp\WObj:=Plywood;
    MoveL Offs(pOrigin,141.15,-142.45,-0.00),v40,z0,tcp\WObj:=Plywood;
    MoveL Offs(pOrigin,142.28,-141.21,-0.00),v40,z0,tcp\WObj:=Plywood;
    MoveL Offs(pOrigin,141.68,-141.53,-0.00),v40,fine,tcp\WObj:=Plywood;
    MoveL Offs(pOrigin,141.68,-141.53,-6.00),v60,z5,tcp\WObj:=Plywood;
    MoveL Offs(pOrigin,147.63,-141.25,-6.00),vTravel,z5,tcp\WObj:=Plywood;
    MoveL Offs(pOrigin,147.63,-141.25,-0.00),v60,z0,tcp\WObj:=Plywood;
    MoveL Offs(pOrigin,148.38,-141.92,-0.00),v40,z0,tcp\WObj:=Plywood;
    MoveL Offs(pOrigin,148.27,-141.53,-0.00),v40,z0,tcp\WObj:=Plywood;
    MoveL Offs(pOrigin,147.63,-141.25,-0.00),v40,z0,tcp\WObj:=Plywood;
    MoveL Offs(pOrigin,148.48,-141.21,-0.00),v40,z0,tcp\WObj:=Plywood;
    MoveL Offs(pOrigin,148.80,-141.57,-0.00),v40,z0,tcp\WObj:=Plywood;
    MoveL Offs(pOrigin,148.98,-140.89,-0.00),v40,z0,tcp\WObj:=Plywood;
    MoveL Offs(pOrigin,148.69,-140.72,-0.00),v40,z0,tcp\WObj:=Plywood;
    MoveL Offs(pOrigin,148.48,-141.21,-0.00),v40,z0,tcp\WObj:=Plywood;
    MoveL Offs(pOrigin,148.48,-140.79,-0.00),v40,z0,tcp\WObj:=Plywood;
    MoveL Offs(pOrigin,148.06,-140.40,-0.00),v40,z0,tcp\WObj:=Plywood;
    MoveL Offs(pOrigin,148.48,-140.79,-0.00),v40,fine,tcp\WObj:=Plywood;
    MoveL Offs(pOrigin,148.48,-140.79,-6.00),v60,z5,tcp\WObj:=Plywood;
    MoveL Offs(pOrigin,148.20,-142.27,-6.00),vTravel,z5,tcp\WObj:=Plywood;
    MoveL Offs(pOrigin,148.20,-142.27,-0.00),v60,z0,tcp\WObj:=Plywood;
    MoveL Offs(pOrigin,148.69,-143.09,-0.00),v40,z0,tcp\WObj:=Plywood;
    MoveL Offs(pOrigin,148.73,-142.70,-0.00),v40,z0,tcp\WObj:=Plywood;
    MoveL Offs(pOrigin,148.20,-142.27,-0.00),v40,fine,tcp\WObj:=Plywood;
    MoveL Offs(pOrigin,148.20,-142.27,-6.00),v60,z5,tcp\WObj:=Plywood;
    MoveL Offs(pOrigin,147.91,-148.86,-6.00),vTravel,z5,tcp\WObj:=Plywood;
    MoveL Offs(pOrigin,147.91,-148.86,-0.00),v60,z0,tcp\WObj:=Plywood;
    MoveL Offs(pOrigin,147.45,-148.33,-0.00),v40,z0,tcp\WObj:=Plywood;
    MoveL Offs(pOrigin,147.91,-148.86,-0.00),v40,fine,tcp\WObj:=Plywood;
    MoveL Offs(pOrigin,147.91,-148.86,-6.00),v60,z5,tcp\WObj:=Plywood;
    MoveL Offs(pOrigin,143.49,-149.75,-6.00),vTravel,z5,tcp\WObj:=Plywood;
  ENDPROC

  PROC DrawPart31()
    MoveL Offs(pOrigin,143.49,-149.75,-0.00),v60,z0,tcp\WObj:=Plywood;
    MoveL Offs(pOrigin,138.39,-153.93,-0.00),v40,z0,tcp\WObj:=Plywood;
    MoveL Offs(pOrigin,140.87,-152.30,-0.00),v40,z0,tcp\WObj:=Plywood;
    MoveL Offs(pOrigin,140.62,-153.11,-0.00),v40,z0,tcp\WObj:=Plywood;
    MoveL Offs(pOrigin,143.49,-149.75,-0.00),v40,fine,tcp\WObj:=Plywood;
    MoveL Offs(pOrigin,143.49,-149.75,-6.00),v60,z5,tcp\WObj:=Plywood;
    MoveL Offs(pOrigin,134.17,-159.06,-6.00),vTravel,z5,tcp\WObj:=Plywood;
    MoveL Offs(pOrigin,134.17,-159.06,-0.00),v60,z0,tcp\WObj:=Plywood;
    MoveL Offs(pOrigin,135.13,-158.96,-0.00),v40,z0,tcp\WObj:=Plywood;
    MoveL Offs(pOrigin,134.17,-159.06,-0.00),v40,fine,tcp\WObj:=Plywood;
    MoveL Offs(pOrigin,134.17,-159.06,-6.00),v60,z5,tcp\WObj:=Plywood;
    MoveL Offs(pOrigin,133.68,-160.44,-6.00),vTravel,z5,tcp\WObj:=Plywood;
    MoveL Offs(pOrigin,133.68,-160.44,-0.00),v60,z0,tcp\WObj:=Plywood;
    MoveL Offs(pOrigin,134.56,-160.87,-0.00),v40,z0,tcp\WObj:=Plywood;
    MoveL Offs(pOrigin,135.55,-160.87,-0.00),v40,z0,tcp\WObj:=Plywood;
    MoveL Offs(pOrigin,133.68,-160.44,-0.00),v40,fine,tcp\WObj:=Plywood;
    MoveL Offs(pOrigin,133.68,-160.44,-6.00),v60,z5,tcp\WObj:=Plywood;
    MoveL Offs(pOrigin,127.76,-161.58,-6.00),vTravel,z5,tcp\WObj:=Plywood;
    MoveL Offs(pOrigin,127.76,-161.58,-0.00),v60,z0,tcp\WObj:=Plywood;
    MoveL Offs(pOrigin,127.34,-161.12,-0.00),v40,z0,tcp\WObj:=Plywood;
    MoveL Offs(pOrigin,127.76,-161.58,-0.00),v40,fine,tcp\WObj:=Plywood;
    MoveL Offs(pOrigin,127.76,-161.58,-6.00),v60,z5,tcp\WObj:=Plywood;
    MoveL Offs(pOrigin,127.05,-170.86,-6.00),vTravel,z5,tcp\WObj:=Plywood;
    MoveL Offs(pOrigin,127.05,-170.86,-0.00),v60,z0,tcp\WObj:=Plywood;
    MoveL Offs(pOrigin,125.07,-171.60,-0.00),v40,z0,tcp\WObj:=Plywood;
    MoveL Offs(pOrigin,126.49,-171.32,-0.00),v40,z0,tcp\WObj:=Plywood;
    MoveL Offs(pOrigin,127.05,-170.86,-0.00),v40,fine,tcp\WObj:=Plywood;
    MoveL Offs(pOrigin,127.05,-170.86,-6.00),v60,z5,tcp\WObj:=Plywood;
    MoveL Offs(pOrigin,131.91,-170.40,-6.00),vTravel,z5,tcp\WObj:=Plywood;
    MoveL Offs(pOrigin,131.91,-170.40,-0.00),v60,z0,tcp\WObj:=Plywood;
    MoveL Offs(pOrigin,133.39,-169.30,-0.00),v40,z0,tcp\WObj:=Plywood;
    MoveL Offs(pOrigin,131.91,-170.40,-0.00),v40,fine,tcp\WObj:=Plywood;
    MoveL Offs(pOrigin,131.91,-170.40,-6.00),v60,z5,tcp\WObj:=Plywood;
    MoveL Offs(pOrigin,117.88,-163.28,-6.00),vTravel,z5,tcp\WObj:=Plywood;
    MoveL Offs(pOrigin,117.88,-163.28,-0.00),v60,z0,tcp\WObj:=Plywood;
    MoveL Offs(pOrigin,117.56,-162.78,-0.00),v40,z0,tcp\WObj:=Plywood;
    MoveL Offs(pOrigin,116.32,-162.25,-0.00),v40,z0,tcp\WObj:=Plywood;
    MoveL Offs(pOrigin,117.14,-163.17,-0.00),v40,z0,tcp\WObj:=Plywood;
    MoveL Offs(pOrigin,117.88,-163.28,-0.00),v40,fine,tcp\WObj:=Plywood;
    MoveL Offs(pOrigin,117.88,-163.28,-6.00),v60,z5,tcp\WObj:=Plywood;
    MoveL Offs(pOrigin,115.65,-162.21,-6.00),vTravel,z5,tcp\WObj:=Plywood;
    MoveL Offs(pOrigin,115.65,-162.21,-0.00),v60,z0,tcp\WObj:=Plywood;
    MoveL Offs(pOrigin,115.01,-160.73,-0.00),v40,z0,tcp\WObj:=Plywood;
    MoveL Offs(pOrigin,114.98,-161.29,-0.00),v40,z0,tcp\WObj:=Plywood;
    MoveL Offs(pOrigin,115.65,-162.21,-0.00),v40,fine,tcp\WObj:=Plywood;
    MoveL Offs(pOrigin,115.65,-162.21,-6.00),v60,z5,tcp\WObj:=Plywood;
    MoveL Offs(pOrigin,112.99,-160.37,-6.00),vTravel,z5,tcp\WObj:=Plywood;
    MoveL Offs(pOrigin,112.99,-160.37,-0.00),v60,z0,tcp\WObj:=Plywood;
    MoveL Offs(pOrigin,113.10,-159.42,-0.00),v40,z0,tcp\WObj:=Plywood;
    MoveL Offs(pOrigin,112.99,-160.37,-0.00),v40,fine,tcp\WObj:=Plywood;
    MoveL Offs(pOrigin,112.99,-160.37,-6.00),v60,z5,tcp\WObj:=Plywood;
    MoveL Offs(pOrigin,109.81,-156.87,-6.00),vTravel,z5,tcp\WObj:=Plywood;
    MoveL Offs(pOrigin,109.81,-156.87,-0.00),v60,z0,tcp\WObj:=Plywood;
    MoveL Offs(pOrigin,108.74,-157.26,-0.00),v40,z0,tcp\WObj:=Plywood;
    MoveL Offs(pOrigin,107.36,-158.92,-0.00),v40,z0,tcp\WObj:=Plywood;
    MoveL Offs(pOrigin,109.81,-156.87,-0.00),v40,fine,tcp\WObj:=Plywood;
    MoveL Offs(pOrigin,109.81,-156.87,-6.00),v60,z5,tcp\WObj:=Plywood;
    MoveL Offs(pOrigin,101.94,-164.91,-6.00),vTravel,z5,tcp\WObj:=Plywood;
    MoveL Offs(pOrigin,101.94,-164.91,-0.00),v60,z0,tcp\WObj:=Plywood;
    MoveL Offs(pOrigin,101.31,-164.62,-0.00),v40,z0,tcp\WObj:=Plywood;
    MoveL Offs(pOrigin,102.90,-167.03,-0.00),v40,z0,tcp\WObj:=Plywood;
    MoveL Offs(pOrigin,103.96,-167.99,-0.00),v40,z0,tcp\WObj:=Plywood;
    MoveL Offs(pOrigin,105.77,-168.84,-0.00),v40,z0,tcp\WObj:=Plywood;
    MoveL Offs(pOrigin,107.22,-168.94,-0.00),v40,z0,tcp\WObj:=Plywood;
    MoveL Offs(pOrigin,104.28,-167.35,-0.00),v40,z0,tcp\WObj:=Plywood;
    MoveL Offs(pOrigin,101.94,-164.91,-0.00),v40,fine,tcp\WObj:=Plywood;
    MoveL Offs(pOrigin,101.94,-164.91,-6.00),v60,z5,tcp\WObj:=Plywood;
    MoveL Offs(pOrigin,105.10,-167.35,-6.00),vTravel,z5,tcp\WObj:=Plywood;
    MoveL Offs(pOrigin,105.10,-167.35,-0.00),v60,z0,tcp\WObj:=Plywood;
    MoveL Offs(pOrigin,107.47,-168.52,-0.00),v40,z0,tcp\WObj:=Plywood;
    MoveL Offs(pOrigin,110.02,-168.94,-0.00),v40,z0,tcp\WObj:=Plywood;
    MoveL Offs(pOrigin,111.93,-168.94,-0.00),v40,z0,tcp\WObj:=Plywood;
    MoveL Offs(pOrigin,113.56,-168.09,-0.00),v40,z0,tcp\WObj:=Plywood;
    MoveL Offs(pOrigin,108.00,-168.20,-0.00),v40,z0,tcp\WObj:=Plywood;
    MoveL Offs(pOrigin,105.10,-167.35,-0.00),v40,fine,tcp\WObj:=Plywood;
    MoveL Offs(pOrigin,105.10,-167.35,-6.00),v60,z5,tcp\WObj:=Plywood;
    MoveL Offs(pOrigin,106.16,-169.26,-6.00),vTravel,z5,tcp\WObj:=Plywood;
    MoveL Offs(pOrigin,106.16,-169.26,-0.00),v60,z0,tcp\WObj:=Plywood;
    MoveL Offs(pOrigin,107.04,-169.58,-0.00),v40,z0,tcp\WObj:=Plywood;
    MoveL Offs(pOrigin,111.12,-169.37,-0.00),v40,z0,tcp\WObj:=Plywood;
    MoveL Offs(pOrigin,108.64,-169.05,-0.00),v40,z0,tcp\WObj:=Plywood;
    MoveL Offs(pOrigin,106.16,-169.26,-0.00),v40,fine,tcp\WObj:=Plywood;
    MoveL Offs(pOrigin,106.16,-169.26,-6.00),v60,z5,tcp\WObj:=Plywood;
    MoveL Offs(pOrigin,97.06,-154.00,-6.00),vTravel,z5,tcp\WObj:=Plywood;
    MoveL Offs(pOrigin,97.06,-154.00,-0.00),v60,z0,tcp\WObj:=Plywood;
    MoveL Offs(pOrigin,96.53,-152.72,-0.00),v40,z0,tcp\WObj:=Plywood;
    MoveL Offs(pOrigin,97.06,-154.00,-0.00),v40,z0,tcp\WObj:=Plywood;
    MoveL Offs(pOrigin,95.89,-153.89,-0.00),v40,z0,tcp\WObj:=Plywood;
    MoveL Offs(pOrigin,95.68,-151.31,-0.00),v40,z0,tcp\WObj:=Plywood;
    MoveL Offs(pOrigin,96.21,-149.18,-0.00),v40,z0,tcp\WObj:=Plywood;
    MoveL Offs(pOrigin,95.78,-148.37,-0.00),v40,z0,tcp\WObj:=Plywood;
    MoveL Offs(pOrigin,95.04,-151.84,-0.00),v40,z0,tcp\WObj:=Plywood;
    MoveL Offs(pOrigin,95.89,-153.89,-0.00),v40,fine,tcp\WObj:=Plywood;
    MoveL Offs(pOrigin,95.89,-153.89,-6.00),v60,z5,tcp\WObj:=Plywood;
    MoveL Offs(pOrigin,97.16,-146.24,-6.00),vTravel,z5,tcp\WObj:=Plywood;
    MoveL Offs(pOrigin,97.16,-146.24,-0.00),v60,z0,tcp\WObj:=Plywood;
    MoveL Offs(pOrigin,96.42,-143.62,-0.00),v40,z0,tcp\WObj:=Plywood;
    MoveL Offs(pOrigin,96.31,-144.82,-0.00),v40,z0,tcp\WObj:=Plywood;
    MoveL Offs(pOrigin,97.16,-146.24,-0.00),v40,fine,tcp\WObj:=Plywood;
    MoveL Offs(pOrigin,97.16,-146.24,-6.00),v60,z5,tcp\WObj:=Plywood;
  ENDPROC

ENDMODULE
